REGION Network 34: PartExist
   RUNG wire#powerrail
      Contact( "AlwaysTRUE" )
      wire#w1
      Contact( "iF-ROOBT3Gripper1Detection" )
      Coil( "KukaRobot3_CtrlDB".sPLCtoROB.User.Gripper.DI133_PartOnGrip1 )
   END_RUNG
   RUNG wire#w1
      Contact( "iF-ROOBT3Gripper2Detection-" )
      Coil( "KukaRobot3_CtrlDB".sPLCtoROB.User.Gripper.DI134_PartOnGrip2 )
   END_RUNG
   // the same network as SCL:
   "KukaRobot3_CtrlDB".sPLCtoROB.User.Gripper.DI133_PartOnGrip1 := "AlwaysTRUE" AND "iF-ROOBT3Gripper1Detection";
   "KukaRobot3_CtrlDB".sPLCtoROB.User.Gripper.DI134_PartOnGrip2 := "AlwaysTRUE" AND "iF-ROOBT3Gripper2Detection-";
END_REGION

REGION Network 35: SpeedCount
   RUNG wire#powerrail
      Contact( "AlwaysTRUE" )
      wire#w1
      { S7_Templates := "SrcType := Int" } GE_Contact(in1 := "Robot_DB".Robot_3.SpeedCount, in2 := 2)
      Coil( "Robot_DB".Robot_3.SpeedChangeFlag )
   END_RUNG
   RUNG wire#w1
      I_Contact( "Station_Sys".Auto.Mode )
      Move(in := 0, out1 => "Robot_DB".Robot_3.SpeedCount)
   END_RUNG
   // the same network as SCL:
   "Robot_DB".Robot_3.SpeedChangeFlag := "AlwaysTRUE" AND ("Robot_DB".Robot_3.SpeedCount >= 2);
   IF "AlwaysTRUE" AND NOT "Station_Sys".Auto.Mode THEN "Robot_DB".Robot_3.SpeedCount := 0; END_IF;
END_REGION

REGION Network 36: Robot3Speed Interlock
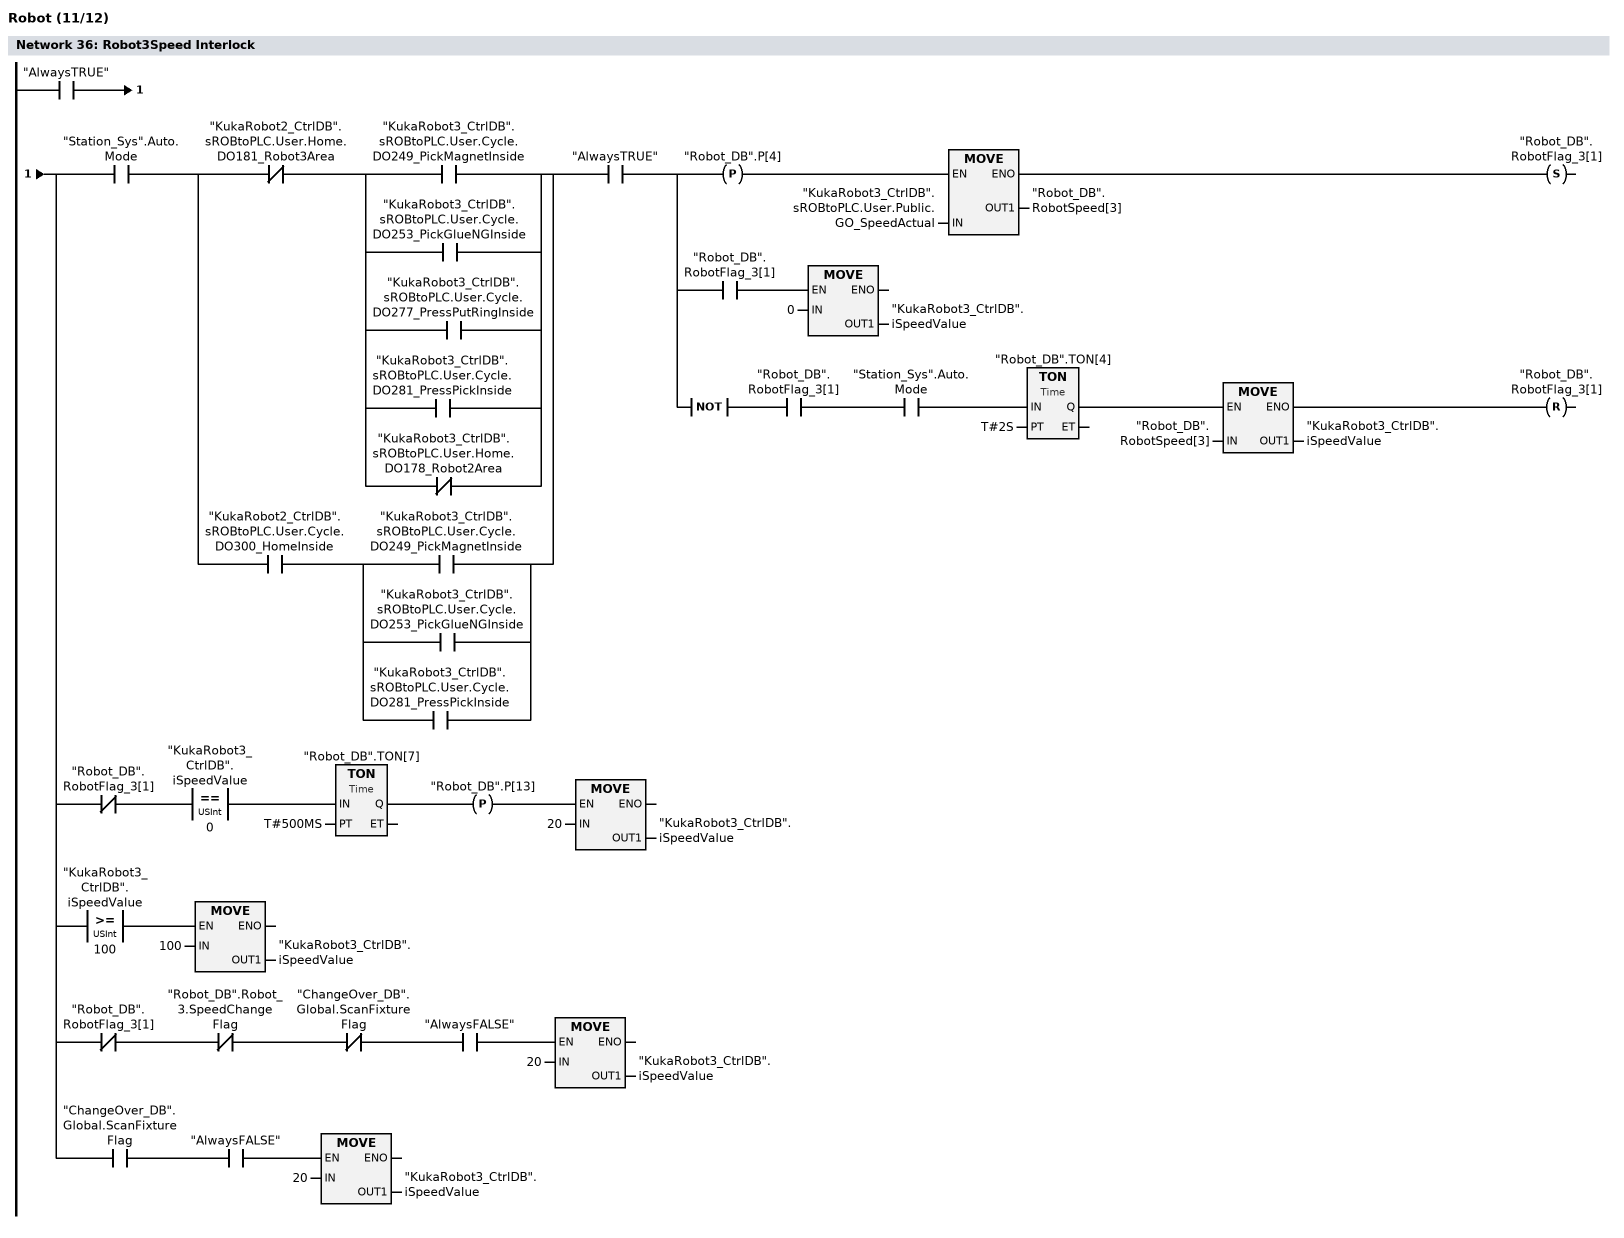
   RUNG wire#powerrail
      Contact( "AlwaysTRUE" )
      wire#w1
      Contact( "Station_Sys".Auto.Mode )
      wire#w2
      I_Contact( "KukaRobot2_CtrlDB".sROBtoPLC.User.Home.DO181_Robot3Area )
      wire#w3
      Contact( "KukaRobot3_CtrlDB".sROBtoPLC.User.Cycle.DO249_PickMagnetInside )
      wire#w4
      Contact( "AlwaysTRUE" )
      wire#w6
      P_Trig( "Robot_DB".P[4] )
      Move(in := "KukaRobot3_CtrlDB".sROBtoPLC.User.Public.GO_SpeedActual, out1 => "Robot_DB".RobotSpeed[3])
      S_Coil( "Robot_DB".RobotFlag_3[1] )
   END_RUNG
   RUNG wire#w3
      Contact( "KukaRobot3_CtrlDB".sROBtoPLC.User.Cycle.DO253_PickGlueNGInside )
   END_RUNG wire#w4
   RUNG wire#w3
      Contact( "KukaRobot3_CtrlDB".sROBtoPLC.User.Cycle.DO277_PressPutRingInside )
   END_RUNG wire#w4
   RUNG wire#w3
      Contact( "KukaRobot3_CtrlDB".sROBtoPLC.User.Cycle.DO281_PressPickInside )
   END_RUNG wire#w4
   RUNG wire#w3
      I_Contact( "KukaRobot3_CtrlDB".sROBtoPLC.User.Home.DO178_Robot2Area )
   END_RUNG wire#w4
   RUNG wire#w2
      Contact( "KukaRobot2_CtrlDB".sROBtoPLC.User.Cycle.DO300_HomeInside )
      wire#w5
      Contact( "KukaRobot3_CtrlDB".sROBtoPLC.User.Cycle.DO249_PickMagnetInside )
   END_RUNG wire#w4
   RUNG wire#w5
      Contact( "KukaRobot3_CtrlDB".sROBtoPLC.User.Cycle.DO253_PickGlueNGInside )
   END_RUNG wire#w4
   RUNG wire#w5
      Contact( "KukaRobot3_CtrlDB".sROBtoPLC.User.Cycle.DO281_PressPickInside )
   END_RUNG wire#w4
   RUNG wire#w6
      Contact( "Robot_DB".RobotFlag_3[1] )
      Move(in := 0, out1 => "KukaRobot3_CtrlDB".iSpeedValue)
   END_RUNG
   RUNG wire#w6
      Not()
      Contact( "Robot_DB".RobotFlag_3[1] )
      Contact( "Station_Sys".Auto.Mode )
      { S7_Templates := "time_type := Time" } "Robot_DB".TON[4].TON(pt := T#2S, et =>)
      Move(in := "Robot_DB".RobotSpeed[3], out1 => "KukaRobot3_CtrlDB".iSpeedValue)
      R_Coil( "Robot_DB".RobotFlag_3[1] )
   END_RUNG
   RUNG wire#w1
      I_Contact( "Robot_DB".RobotFlag_3[1] )
      { S7_Templates := "SrcType := USInt" } EQ_Contact(in1 := "KukaRobot3_CtrlDB".iSpeedValue, in2 := 0)
      { S7_Templates := "time_type := Time" } "Robot_DB".TON[7].TON(pt := T#500MS, et =>)
      P_Trig( "Robot_DB".P[13] )
      Move(in := 20, out1 => "KukaRobot3_CtrlDB".iSpeedValue)
   END_RUNG
   RUNG wire#w1
      { S7_Templates := "SrcType := USInt" } GE_Contact(in1 := "KukaRobot3_CtrlDB".iSpeedValue, in2 := 100)
      Move(in := 100, out1 => "KukaRobot3_CtrlDB".iSpeedValue)
   END_RUNG
   RUNG wire#w1
      I_Contact( "Robot_DB".RobotFlag_3[1] )
      I_Contact( "Robot_DB".Robot_3.SpeedChangeFlag )
      I_Contact( "ChangeOver_DB".Global.ScanFixtureFlag )
      Contact( "AlwaysFALSE" )
      Move(in := 20, out1 => "KukaRobot3_CtrlDB".iSpeedValue)
   END_RUNG
   RUNG wire#w1
      Contact( "ChangeOver_DB".Global.ScanFixtureFlag )
      Contact( "AlwaysFALSE" )
      Move(in := 20, out1 => "KukaRobot3_CtrlDB".iSpeedValue)
   END_RUNG
   // the same network as SCL:
   #_w1 := "AlwaysTRUE" AND "Station_Sys".Auto.Mode AND ((NOT "KukaRobot2_CtrlDB".sROBtoPLC.User.Home.DO181_Robot3Area AND ("KukaRobot3_CtrlDB".sROBtoPLC.User.Cycle.DO249_PickMagnetInside OR "KukaRobot3_CtrlDB".sROBtoPLC.User.Cycle.DO253_PickGlueNGInside OR "KukaRobot3_CtrlDB".sROBtoPLC.User.Cycle.DO277_PressPutRingInside OR "KukaRobot3_CtrlDB".sROBtoPLC.User.Cycle.DO281_PressPickInside OR NOT "KukaRobot3_CtrlDB".sROBtoPLC.User.Home.DO178_Robot2Area)) OR ("KukaRobot2_CtrlDB".sROBtoPLC.User.Cycle.DO300_HomeInside AND ("KukaRobot3_CtrlDB".sROBtoPLC.User.Cycle.DO249_PickMagnetInside OR "KukaRobot3_CtrlDB".sROBtoPLC.User.Cycle.DO253_PickGlueNGInside OR "KukaRobot3_CtrlDB".sROBtoPLC.User.Cycle.DO281_PressPickInside))) AND "AlwaysTRUE";
   #_w2 := #_w1 AND NOT "Robot_DB".P[4];   // rising edge
   "Robot_DB".P[4] := #_w1;
   IF #_w2 THEN
       "Robot_DB".RobotSpeed[3] := "KukaRobot3_CtrlDB".sROBtoPLC.User.Public.GO_SpeedActual;
       "Robot_DB".RobotFlag_3[1] := TRUE;
   END_IF;
   IF #_w1 AND "Robot_DB".RobotFlag_3[1] THEN "KukaRobot3_CtrlDB".iSpeedValue := 0; END_IF;
   "Robot_DB".TON[4].TON(IN := NOT #_w1 AND "Robot_DB".RobotFlag_3[1] AND "Station_Sys".Auto.Mode, PT := T#2S);
   IF "Robot_DB".TON[4].Q THEN
       "KukaRobot3_CtrlDB".iSpeedValue := "Robot_DB".RobotSpeed[3];
       "Robot_DB".RobotFlag_3[1] := FALSE;
   END_IF;
   "Robot_DB".TON[7].TON(IN := "AlwaysTRUE" AND NOT "Robot_DB".RobotFlag_3[1] AND ("KukaRobot3_CtrlDB".iSpeedValue = 0),
                         PT := T#500MS);
   #_w3 := "Robot_DB".TON[7].Q AND NOT "Robot_DB".P[13];   // rising edge
   "Robot_DB".P[13] := "Robot_DB".TON[7].Q;
   IF #_w3 THEN "KukaRobot3_CtrlDB".iSpeedValue := 20; END_IF;
   IF "AlwaysTRUE" AND ("KukaRobot3_CtrlDB".iSpeedValue >= 100) THEN
       "KukaRobot3_CtrlDB".iSpeedValue := 100;
   END_IF;
   IF "AlwaysTRUE" AND NOT "Robot_DB".RobotFlag_3[1] AND NOT "Robot_DB".Robot_3.SpeedChangeFlag AND NOT "ChangeOver_DB".Global.ScanFixtureFlag AND "AlwaysFALSE" THEN
       "KukaRobot3_CtrlDB".iSpeedValue := 20;
   END_IF;
   IF "AlwaysTRUE" AND "ChangeOver_DB".Global.ScanFixtureFlag AND "AlwaysFALSE" THEN
       "KukaRobot3_CtrlDB".iSpeedValue := 20;
   END_IF;
END_REGION

REGION Network 37: Robot3 No Task Running
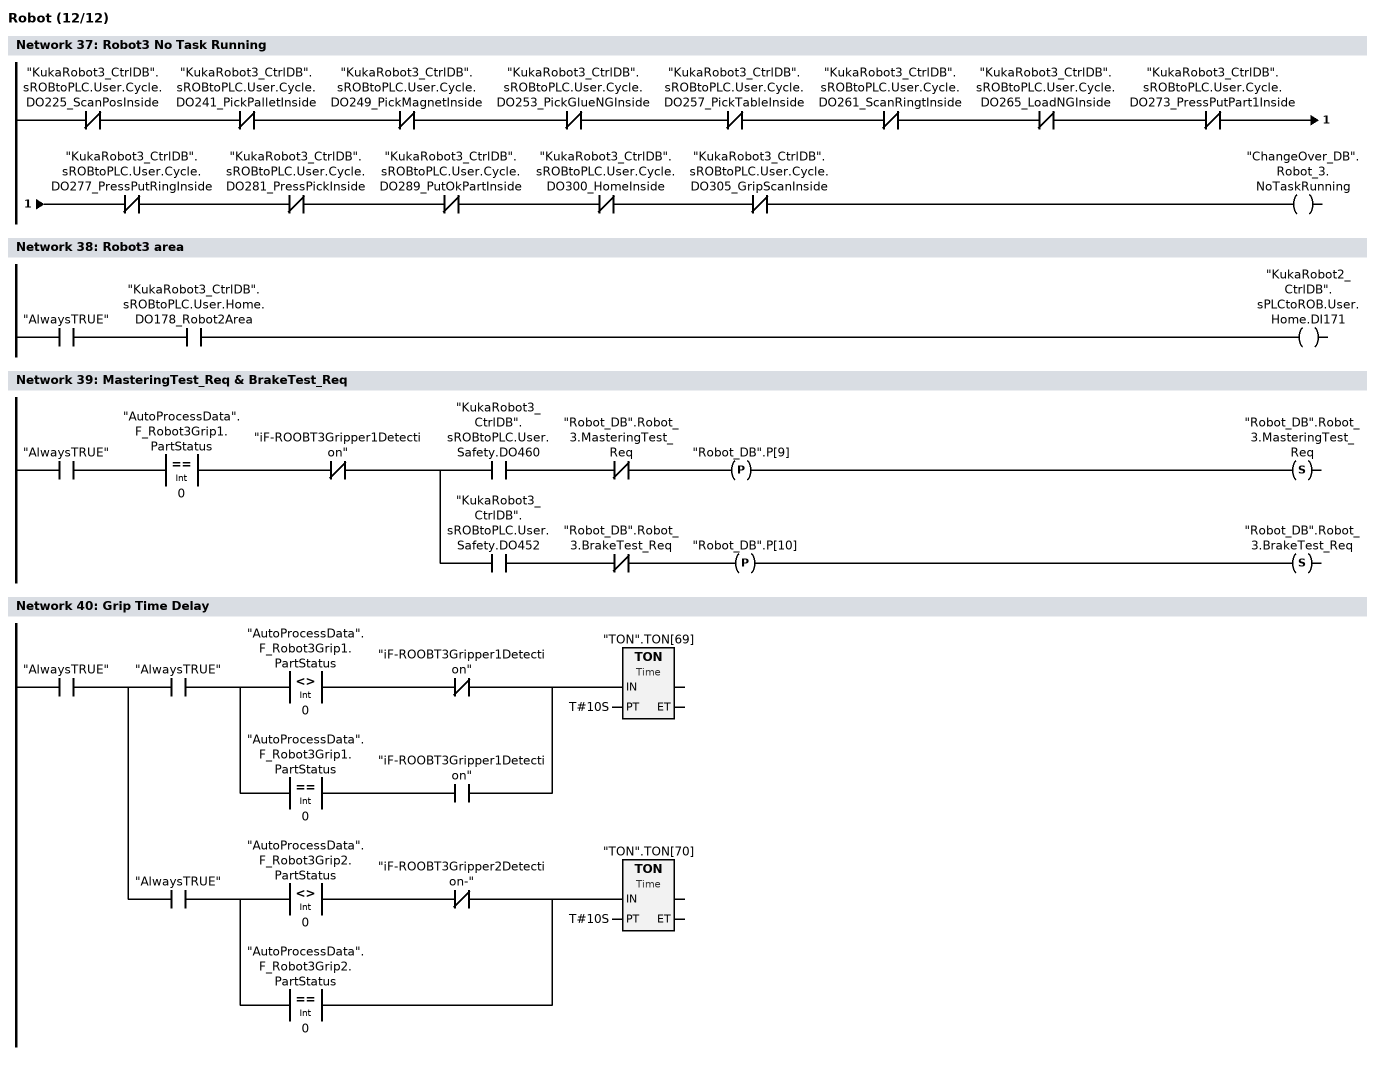
   RUNG wire#powerrail
      I_Contact( "KukaRobot3_CtrlDB".sROBtoPLC.User.Cycle.DO225_ScanPosInside )
      I_Contact( "KukaRobot3_CtrlDB".sROBtoPLC.User.Cycle.DO241_PickPalletInside )
      I_Contact( "KukaRobot3_CtrlDB".sROBtoPLC.User.Cycle.DO249_PickMagnetInside )
      I_Contact( "KukaRobot3_CtrlDB".sROBtoPLC.User.Cycle.DO253_PickGlueNGInside )
      I_Contact( "KukaRobot3_CtrlDB".sROBtoPLC.User.Cycle.DO257_PickTableInside )
      I_Contact( "KukaRobot3_CtrlDB".sROBtoPLC.User.Cycle.DO261_ScanRingtInside )
      I_Contact( "KukaRobot3_CtrlDB".sROBtoPLC.User.Cycle.DO265_LoadNGInside )
      I_Contact( "KukaRobot3_CtrlDB".sROBtoPLC.User.Cycle.DO273_PressPutPart1Inside )
      I_Contact( "KukaRobot3_CtrlDB".sROBtoPLC.User.Cycle.DO277_PressPutRingInside )
      I_Contact( "KukaRobot3_CtrlDB".sROBtoPLC.User.Cycle.DO281_PressPickInside )
      I_Contact( "KukaRobot3_CtrlDB".sROBtoPLC.User.Cycle.DO289_PutOkPartInside )
      I_Contact( "KukaRobot3_CtrlDB".sROBtoPLC.User.Cycle.DO300_HomeInside )
      I_Contact( "KukaRobot3_CtrlDB".sROBtoPLC.User.Cycle.DO305_GripScanInside )
      Coil( "ChangeOver_DB".Robot_3.NoTaskRunning )
   END_RUNG
   // the same network as SCL:
   "ChangeOver_DB".Robot_3.NoTaskRunning := NOT "KukaRobot3_CtrlDB".sROBtoPLC.User.Cycle.DO225_ScanPosInside AND NOT "KukaRobot3_CtrlDB".sROBtoPLC.User.Cycle.DO241_PickPalletInside AND NOT "KukaRobot3_CtrlDB".sROBtoPLC.User.Cycle.DO249_PickMagnetInside AND NOT "KukaRobot3_CtrlDB".sROBtoPLC.User.Cycle.DO253_PickGlueNGInside AND NOT "KukaRobot3_CtrlDB".sROBtoPLC.User.Cycle.DO257_PickTableInside AND NOT "KukaRobot3_CtrlDB".sROBtoPLC.User.Cycle.DO261_ScanRingtInside AND NOT "KukaRobot3_CtrlDB".sROBtoPLC.User.Cycle.DO265_LoadNGInside AND NOT "KukaRobot3_CtrlDB".sROBtoPLC.User.Cycle.DO273_PressPutPart1Inside AND NOT "KukaRobot3_CtrlDB".sROBtoPLC.User.Cycle.DO277_PressPutRingInside AND NOT "KukaRobot3_CtrlDB".sROBtoPLC.User.Cycle.DO281_PressPickInside AND NOT "KukaRobot3_CtrlDB".sROBtoPLC.User.Cycle.DO289_PutOkPartInside AND NOT "KukaRobot3_CtrlDB".sROBtoPLC.User.Cycle.DO300_HomeInside AND NOT "KukaRobot3_CtrlDB".sROBtoPLC.User.Cycle.DO305_GripScanInside;
END_REGION

REGION Network 38: Robot3 area
   RUNG wire#powerrail
      Contact( "AlwaysTRUE" )
      Contact( "KukaRobot3_CtrlDB".sROBtoPLC.User.Home.DO178_Robot2Area )
      Coil( "KukaRobot2_CtrlDB".sPLCtoROB.User.Home.DI171 )
   END_RUNG
   // the same network as SCL:
   "KukaRobot2_CtrlDB".sPLCtoROB.User.Home.DI171 := "AlwaysTRUE" AND "KukaRobot3_CtrlDB".sROBtoPLC.User.Home.DO178_Robot2Area;
END_REGION

REGION Network 39: MasteringTest_Req & BrakeTest_Req
   RUNG wire#powerrail
      Contact( "AlwaysTRUE" )
      { S7_Templates := "SrcType := Int" } EQ_Contact(in1 := "AutoProcessData".F_Robot3Grip1.PartStatus, in2 := 0)
      I_Contact( "iF-ROOBT3Gripper1Detection" )
      wire#w1
      Contact( "KukaRobot3_CtrlDB".sROBtoPLC.User.Safety.DO460 )
      I_Contact( "Robot_DB".Robot_3.MasteringTest_Req )
      P_Trig( "Robot_DB".P[9] )
      S_Coil( "Robot_DB".Robot_3.MasteringTest_Req )
   END_RUNG
   RUNG wire#w1
      Contact( "KukaRobot3_CtrlDB".sROBtoPLC.User.Safety.DO452 )
      I_Contact( "Robot_DB".Robot_3.BrakeTest_Req )
      P_Trig( "Robot_DB".P[10] )
      S_Coil( "Robot_DB".Robot_3.BrakeTest_Req )
   END_RUNG
   // the same network as SCL:
   #_w1 := "AlwaysTRUE" AND ("AutoProcessData".F_Robot3Grip1.PartStatus = 0) AND NOT "iF-ROOBT3Gripper1Detection";
   #_w2 := #_w1 AND "KukaRobot3_CtrlDB".sROBtoPLC.User.Safety.DO460 AND NOT "Robot_DB".Robot_3.MasteringTest_Req;
   #_w3 := #_w2 AND NOT "Robot_DB".P[9];   // rising edge
   "Robot_DB".P[9] := #_w2;
   IF #_w3 THEN "Robot_DB".Robot_3.MasteringTest_Req := TRUE; END_IF;
   #_w4 := #_w1 AND "KukaRobot3_CtrlDB".sROBtoPLC.User.Safety.DO452 AND NOT "Robot_DB".Robot_3.BrakeTest_Req;
   #_w5 := #_w4 AND NOT "Robot_DB".P[10];   // rising edge
   "Robot_DB".P[10] := #_w4;
   IF #_w5 THEN "Robot_DB".Robot_3.BrakeTest_Req := TRUE; END_IF;
END_REGION

REGION Network 40: Grip Time Delay
   RUNG wire#powerrail
      Contact( "AlwaysTRUE" )
      wire#w1
      Contact( "AlwaysTRUE" )
      wire#w2
      { S7_Templates := "SrcType := Int" } NE_Contact(in1 := "AutoProcessData".F_Robot3Grip1.PartStatus, in2 := 0)
      I_Contact( "iF-ROOBT3Gripper1Detection" )
      wire#w3
      { S7_Templates := "time_type := Time" } "TON".TON[69].TON(pt := T#10S, et =>)
   END_RUNG
   RUNG wire#w2
      { S7_Templates := "SrcType := Int" } EQ_Contact(in1 := "AutoProcessData".F_Robot3Grip1.PartStatus, in2 := 0)
      Contact( "iF-ROOBT3Gripper1Detection" )
   END_RUNG wire#w3
   RUNG wire#w1
      Contact( "AlwaysTRUE" )
      wire#w4
      { S7_Templates := "SrcType := Int" } NE_Contact(in1 := "AutoProcessData".F_Robot3Grip2.PartStatus, in2 := 0)
      I_Contact( "iF-ROOBT3Gripper2Detection-" )
      wire#w5
      { S7_Templates := "time_type := Time" } "TON".TON[70].TON(pt := T#10S, et =>)
   END_RUNG
   RUNG wire#w4
      { S7_Templates := "SrcType := Int" } EQ_Contact(in1 := "AutoProcessData".F_Robot3Grip2.PartStatus, in2 := 0)
   END_RUNG wire#w5
   // the same network as SCL:
   "TON".TON[69].TON(IN := "AlwaysTRUE" AND "AlwaysTRUE" AND ((("AutoProcessData".F_Robot3Grip1.PartStatus <> 0) AND NOT "iF-ROOBT3Gripper1Detection") OR (("AutoProcessData".F_Robot3Grip1.PartStatus = 0) AND "iF-ROOBT3Gripper1Detection")),
                     PT := T#10S);
   "TON".TON[70].TON(IN := "AlwaysTRUE" AND "AlwaysTRUE" AND ((("AutoProcessData".F_Robot3Grip2.PartStatus <> 0) AND NOT "iF-ROOBT3Gripper2Detection-") OR ("AutoProcessData".F_Robot3Grip2.PartStatus = 0)),
                     PT := T#10S);
END_REGION
END_FUNCTION

FUNCTION_BLOCK "KukaRobot1_Ctrl"   // FB2401, SCL
{ S7_Optimized_Access := 'FALSE' }
// stored: AutoNumber false, SetENOAutomatically false
   VAR_INPUT
      iHWID_In : HW_IO;
      iHWID_Out : HW_IO;
      iSysRun : Bool;
      iAuto : Bool;
      iManual : Bool;
      iSpecial : Bool;
      iE_STOP : Bool;
      iReset : Bool;
      iT1000ms : Bool;
      iTaskMode : USInt;
      iPartType : USInt;
      iSpeedValue : USInt;
      iPGNO : USInt;   // Robot Program number
   END_VAR
   VAR_OUTPUT
      oReady : Bool;
      oStartComplete : Bool;
      oWarning : Bool;
      oError : Bool;
      oErrorCode : Int;
   END_VAR
   VAR_IN_OUT
      ioAutoStart : Bool;
      ioSrartHome : Bool;
      ioStartAutoCycle : Bool;
   END_VAR
   VAR
      sHMI { S7_SetPoint := 'True'} : "KukaRobot_HMI";
      sROBtoPLC : Struct
         Sys { S7_SetPoint := 'True'} : "KukaRobot_SysOutput";   // Robot ---> PLC
         User { S7_SetPoint := 'True'} : "KukaRobot_UserOutput_1";   // Robot ---> PLC
      END_STRUCT;
      sPLCtoROB : Struct
         Sys { S7_SetPoint := 'True'} : "KukaRobot_SysInput";   // PLC ---> Robot
         User { S7_SetPoint := 'True'} : "KukaRobot_UserInput_1";   // PLC ---> Robot
      END_STRUCT;
      sDrivesOnDelay { S7_SetPoint := 'True'} : TON_TIME;
      sStartUpDelay { S7_SetPoint := 'True'} : TON_TIME;
      sRobotReadyToStart : Bool;
      sRobotReadyToRunning : Bool;
      sRobotActComplete : Bool;
      sRobotProgrameChoseOK : Bool;
      sSequence : Int;
      F_TRIG_Work { S7_SetPoint := 'True'} : F_TRIG;
      F_TRIG_Home { S7_SetPoint := 'True'} : F_TRIG;
      ModeValue : Int;
      Tem_ModeValue : Int;
      ModeChange : Bool;
      IEC_Timer_DRIVES_OFF { S7_SetPoint := 'True'} : TON_TIME;
      IEC_Timer_DRIVES_ON { S7_SetPoint := 'True'} : TON_TIME;
   END_VAR
   VAR_TEMP
      tInRwENO : Bool;
      tOutRwENO : Bool;
      tInRwRetVal : Int;
      tOutRwRetVal : Int;
      "tROB-Input" : Array[1..128] of Byte;
      tROB_Output : Array[1..128] of Byte;
   END_VAR
BEGIN
   REGION Description
       (*
       %%%
   VERSION: V1.0
   LANGUAGE: ENGLISH
       %%%
       ** ** ** ** ** ** ** ** ** ** ** ** ** ** ** ** ** ** ** ** ** ** ** ** ** ** ** ** ** ** ** ** ** ** ** ** ** ** ** ** ** ** ** ** ** ** ** ** ** **
       ** ** ** ** ** ** ** ** ** ** ** ** ** ** ** ** ** ** ** ** ** ** ** ** ** ** ** ** ** ** ** ** ** ** ** ** ** ** ** ** ** ** ** ** ** ** ** ** ** **
       * *
       * R (uhlamat) R (obot) I (nterface) *
       * < < Robot Function Block > > *
       * < < Handing Tool > > *
       * - - - - - - - - - - - - - - - - - - - - - - - - - - - - - - - - - - - - - - - - - - *
       * *
       * Customer:   *
       * Roboter Type: Kuka *
       * Software: Siemens TIA V15.1 SP1 *
       * Autor: ChenYi *
       * Company: Ruhlamat Automation Technologies (Suzhou) Co., Ltd *
       * Department: Elec.*
       * Telephone: + 86 (512) 6767 1108 *
       * *
       * Version: 1.0 *
       * Created: 26.05.2020 *
       * Modified: 26.05.2020
   BY: ChenYi *
       * *
       ** ** ** ** ** ** ** ** ** ** ** ** ** ** ** ** ** ** ** ** ** ** ** ** ** ** ** ** ** ** ** ** ** ** ** ** ** ** ** ** ** ** ** ** ** ** ** ** ** **
       ** ** ** ** ** ** ** ** ** ** ** ** ** ** ** ** ** ** ** ** ** ** ** ** ** ** ** ** ** ** ** ** ** ** ** ** ** ** ** ** ** ** ** ** ** ** ** ** ** **
       %%%
    #oErrorCode:
       102:Robot home Failed
       205:Failed to read HW Input data;
       206:Failed to write HW Output data;
       303:Start up TimeOut   

       %%%
       *)
   END_REGION
   //<<<<<<<<<<<<<<<<<<<<<<<<<<<<<<<<<<<<<<<<<<<<<<<<<>>>>>>>>>>>>>>>>>>>>>>>>>>>>>>>>>>>>>>>>>>>>>>>>>
   //<<<<<<<<<<<<<<<<<<<<<<<<<<<<<<<<<<<<<<<<  Program Start  >>>>>>>>>>>>>>>>>>>>>>>>>>>>>>>>>>>>>>>>>
   //<<<<<<<<<<<<<<<<<<<<<<<<<<<<<<<<<<<<<<<<<<<<<<<<<>>>>>>>>>>>>>>>>>>>>>>>>>>>>>>>>>>>>>>>>>>>>>>>>>




   //******************************************
   REGION Bus Input Data Mapping

       #tInRwRetVal := DPRD_DAT(LADDR := #iHWID_In, RECORD => #sROBtoPLC, ENO => #tInRwENO);
       IF NOT #tInRwENO THEN
           GOTO ERROR;
       END_IF;

   END_REGION


   //******************************************
   (*Robot controller remmote control*)

   // I/O Act-Activate interface
   #sPLCtoROB.Sys.SI.I_O_ACT := 1;
   // Move Enable
   //#sPLCtoROB.Sys.SI.MOVE_ENABLE := (#iSysRun AND (((#sROBtoPLC.Sys.SO.T1 OR #sROBtoPLC.Sys.SO.T2) AND #iManual) OR (#iAuto))) AND #iSafePos;
   //#sPLCtoROB.Sys.SI.MOVE_ENABLE := #iSysRun AND (#iManual OR #iAuto) AND #iSafePos;
   IF #sROBtoPLC.Sys.SO.EXT = TRUE THEN
       #sPLCtoROB.Sys.SI.MOVE_ENABLE := #iE_STOP;
   END_IF;
   IF #sROBtoPLC.Sys.SO.T1 = TRUE OR #sROBtoPLC.Sys.SO.T2 = TRUE THEN
       #sPLCtoROB.Sys.SI.MOVE_ENABLE := TRUE;
   END_IF;
   // Drives Off
   #sPLCtoROB.Sys.SI.DRIVES_OFF := NOT #ModeChange;


   IF #iManual
   THEN
       #ModeValue := 1;
   ELSIF #iAuto
   THEN
       #ModeValue := 3;

   END_IF;

   IF #ModeValue <> #Tem_ModeValue
   THEN
       #ModeChange := true;
   ELSE
       #ModeChange := false;
   END_IF;

   IF #IEC_Timer_DRIVES_OFF.Q THEN
       #Tem_ModeValue := #ModeValue;
   END_IF;

   #IEC_Timer_DRIVES_OFF(IN:=#ModeValue <> #Tem_ModeValue,
                         PT:=T#1s);


   //#sPLCtoROB.Sys.SI.DRIVES_OFF := #iSysRun;
   //#sPLCtoROB.Sys.SI.DRIVES_OFF := #iSysRun AND (#iManual OR #iAuto) AND #iSafePos;
   (*Robot controller ready to Start*)
   #sRobotReadyToStart := #iSysRun AND (#iAuto OR #iSpecial) AND
   #sROBtoPLC.Sys.SO.USER_SAF AND #sROBtoPLC.Sys.SO.ALARM_STOP AND
   #sROBtoPLC.Sys.SO.I_O_ACTCONF AND #sROBtoPLC.Sys.SO.ALARM_STOP_INTERN AND
   #sPLCtoROB.Sys.SI.MOVE_ENABLE AND #sPLCtoROB.Sys.SI.DRIVES_OFF
   AND #sROBtoPLC.Sys.SO.EXT;


   REGION Robot Start control
       IF #sRobotReadyToStart THEN
           IF (#sSequence = 0) AND #ioAutoStart AND (#iAuto OR #iSpecial) AND NOT #sRobotActComplete THEN
               #sSequence := 100;
               #ioAutoStart := 0;
               #sRobotActComplete := 0;
               #sRobotProgrameChoseOK := 0;
           END_IF;

           #IEC_Timer_DRIVES_ON(IN := #sSequence=110,
                                 PT := T#100ms);

           CASE #sSequence OF
   (*            100:
                   #sPLCtoROB.Sys.SI.DRIVES_ON := 0;
                   #sSequence := 110;

               110:
                   #sPLCtoROB.Sys.SI.DRIVES_ON := 1;
                   IF #IEC_Timer_DRIVES_ON.Q THEN
                       #sPLCtoROB.Sys.SI.DRIVES_ON := 0;
                       #sSequence := 150;
                   END_IF;
                   *)
               100:  // DrivesOn
                   IF NOT #sROBtoPLC.Sys.SO.RC_RDY1  THEN
                           #sPLCtoROB.Sys.SI.CONF_MESS := 1;
                           #sPLCtoROB.Sys.SI.DRIVES_ON := 0;
                       ELSIF #sROBtoPLC.Sys.SO.RC_RDY1 THEN
                           #sPLCtoROB.Sys.SI.CONF_MESS := 0;
                           #sPLCtoROB.Sys.SI.DRIVES_ON := 1;
                           IF #sDrivesOnDelay.Q AND #sROBtoPLC.Sys.SO.PERI_RDY THEN
                               #sSequence := 200;
                               #sPLCtoROB.Sys.SI.DRIVES_ON := 0;

                           END_IF;
                       END_IF;

                       200:  // ALARM CONF
                       IF #sROBtoPLC.Sys.SO.STOPMESS OR NOT #sROBtoPLC.Sys.SO.RC_RDY1 THEN
                           #sPLCtoROB.Sys.SI.CONF_MESS := 1;
                       ELSE
                           #sPLCtoROB.Sys.SI.CONF_MESS := 0;
                           #sSequence := 300;
                       END_IF;

                       300: // EXT_Start    
                       IF #sROBtoPLC.Sys.SO.PERI_RDY AND NOT #sROBtoPLC.Sys.SO.STOPMESS THEN
                           #sPLCtoROB.Sys.SI.EXT_START := 1;
                           #sSequence := 400;
                       END_IF;

                       400: // EXT_Start Reset  
                       IF #sROBtoPLC.Sys.SO.PRO_ACT THEN
                           #sPLCtoROB.Sys.SI.EXT_START := 0;
                           #sSequence := 500;
                       END_IF;

                       500: // Programe Call
                       IF #sROBtoPLC.Sys.SO.PERI_RDY
                           AND #sROBtoPLC.Sys.SO.PRO_ACT
                           AND #sROBtoPLC.Sys.SO.PGNO_REQ
                           AND #iPGNO <> 0
                           //AND #s_ROBInput.User.User.Home.DI_AutoCycleStart
                           //AND #s_ROBOutput.Sys."SO_$ON_PATH"
                           //AND #s_ROBOutput.Sys."SO_$IN_HOME"
                       THEN

                           #sPLCtoROB.Sys.SI.PGNO_PBIT := #iPGNO;
                           #sPLCtoROB.Sys.SI.PGNO_VALID := 1;
                           #sSequence := 600;
                       END_IF;

                       600: // Programe Call Finish
                       IF #sROBtoPLC.Sys.SO.APPL_RUN THEN
                           #sPLCtoROB.Sys.SI.PGNO_VALID := 0;
                           #sRobotActComplete := 1;
                           #sSequence := 0;
                       END_IF;

           END_CASE;

       ELSE
           #sSequence := 0;
           #sRobotActComplete := 0;
   //        #sPLCtoROB.Sys.SI.DRIVES_ON := 0;////2023/9/1更改
           #sPLCtoROB.Sys.SI.EXT_START := 0;
          // #sPLCtoROB.Sys.SI.CONF_MESS := 0;
           #sPLCtoROB.Sys.SI.PGNO_VALID := 0;
           #sPLCtoROB.Sys.SI.PGNO_PBIT := 0; 
       END_IF;

   (*Robot ready to Running*)
       #sRobotReadyToRunning := #sRobotReadyToStart AND #sROBtoPLC.Sys.SO.PERI_RDY AND #sROBtoPLC.Sys.SO.PRO_ACT AND #sROBtoPLC.Sys.SO.APPL_RUN;


   (*Robot TaskMode,PartType, SpeedValue Set*)
       #sPLCtoROB.User.Public.GI_TaskMode := #iTaskMode;
       #sPLCtoROB.User.Public.GI_PartType := #iPartType;
       #sPLCtoROB.User.Public.GI_SpeedSet := #iSpeedValue;

       // Robot Program calls
       #sPLCtoROB.Sys.SI.PGNO_PARITY := 1;
       //************************************************************
       (*DrivesOn delay*)
       #sDrivesOnDelay(IN := #sPLCtoROB.Sys.SI.DRIVES_ON,
                       PT := T#200ms      // IN: TIME
       );
   (*StartTimeOut delay*)
       #sStartUpDelay(IN := #sSequence <> 0,
                      PT := T#5s        // IN: TIME
       );
       IF #sStartUpDelay.Q THEN
           #sHMI.StartUpTimeOut := 1;
           GOTO ERROR;
       ELSE
           #sHMI.StartUpTimeOut := 0;
       END_IF;

   END_REGION

   //******************************************
   REGION Home
       IF #sRobotReadyToRunning AND #sROBtoPLC.User.Home.DO161_WaitForHomeSeqStart AND NOT #sROBtoPLC.User.Home.DO162_GoHomeFail AND #ioSrartHome THEN
           #sPLCtoROB.User.Home.DI161_HomeSeqStart := 1;
       END_IF;

       IF #sRobotReadyToRunning AND #sROBtoPLC.User.Home.DO163_HomeSeqOK THEN
           #ioSrartHome := 0;
           #sPLCtoROB.User.Home.DI161_HomeSeqStart := 0;
       END_IF;

       IF #sROBtoPLC.User.Home.DO162_GoHomeFail THEN
           GOTO ERROR;
       END_IF;

   END_REGION ;

   REGION Auto Cycle Start

       (*Start Auto Cycle*)
       IF #sRobotReadyToRunning AND #sROBtoPLC.User.Home.DO164_WaitForAutoStart AND #ioStartAutoCycle THEN
           #sPLCtoROB.User.Home.DI162_AutoCycleStart := 1;
       ELSE
           #sPLCtoROB.User.Home.DI162_AutoCycleStart := 0;
       END_IF;

       IF NOT #sROBtoPLC.User.Home.DO164_WaitForAutoStart THEN
           #ioStartAutoCycle := 0;
       END_IF;


   END_REGION ;




   REGION Bus Output Data Mapping

       #tOutRwRetVal := DPWR_DAT(LADDR := #iHWID_Out, RECORD := #sPLCtoROB, ENO => #tOutRwENO);
       IF NOT #tOutRwENO THEN
           GOTO ERROR;
       END_IF;

   END_REGION

   //----------------------------------------------------------------------------------------------------
   REGION Output
       #oReady := #sRobotReadyToRunning;
       #oStartComplete := #sRobotActComplete;


   END_REGION

   REGION HMI Signal
       //SI  
       #sHMI.PGNO_PBIT := #sPLCtoROB.Sys.SI.PGNO_PBIT;
       #sHMI.EXT_START := #sPLCtoROB.Sys.SI.EXT_START;
       #sHMI.MOVE_ENABLE := #sHMI.MOVE_ENABLE;
       #sHMI.CONF_MESS := #sPLCtoROB.Sys.SI.CONF_MESS;
       #sHMI.DRIVES_OFF := NOT #sHMI.DRIVES_OFF;
       #sHMI.DRIVES_ON := #sHMI.DRIVES_ON;
       #sHMI.I_O_ACT := #sHMI.I_O_ACT;
       //UI   
       #sHMI.TaskMode := #sPLCtoROB.User.Public.GI_TaskMode;
       #sHMI.PartType := #sPLCtoROB.User.Public.GI_PartType;
       #sHMI.SpeedSet := #sPLCtoROB.User.Public.GI_SpeedSet;
       #sHMI.HomeSeqStart := #sPLCtoROB.User.Home.DI161_HomeSeqStart;
       #sHMI.AutoCycleStart := #sPLCtoROB.User.Home.DI162_AutoCycleStart;
       //SO   
       #sHMI.RC_RDY1 := #sROBtoPLC.Sys.SO.RC_RDY1;
       #sHMI.ALARM_STOP := NOT #sROBtoPLC.Sys.SO.ALARM_STOP;
       #sHMI.USER_SAF := #sROBtoPLC.Sys.SO.USER_SAF;
       #sHMI.PERI_RDY := #sROBtoPLC.Sys.SO.PERI_RDY;
       #sHMI.ROB_CAL := #sROBtoPLC.Sys.SO.ROB_CAL;
       #sHMI.I_O_ACTCONF := #sROBtoPLC.Sys.SO.I_O_ACTCONF;
       #sHMI.STOPMESS := #sROBtoPLC.Sys.SO.STOPMESS;
       #sHMI.ALARM_STOP_INTERN := NOT #sROBtoPLC.Sys.SO.ALARM_STOP_INTERN;
       #sHMI.PGNO_FBIT_REFL := #sROBtoPLC.Sys.SO.PGNO_FBIT_REFL;
       #sHMI.PRO_ACT := #sROBtoPLC.Sys.SO.PRO_ACT;
       #sHMI.APPL_RUN := #sROBtoPLC.Sys.SO.APPL_RUN;
       #sHMI.PRO_MOVE := #sROBtoPLC.Sys.SO.PRO_MOVE;
       #sHMI.IN_HOME := #sROBtoPLC.Sys.SO.IN_HOME;
       #sHMI.ON_PATH := #sROBtoPLC.Sys.SO.ON_PATH;
       #sHMI.NEAR_POSRET := #sROBtoPLC.Sys.SO.NEAR_POSRET;
       #sHMI.T1 := #sROBtoPLC.Sys.SO.T1;
       #sHMI.T2 := #sROBtoPLC.Sys.SO.T2;
       #sHMI.AUT := #sROBtoPLC.Sys.SO.AUT;
       #sHMI.EXT := #sROBtoPLC.Sys.SO.EXT;
       //UO
       #sHMI.CurrentMode := #sROBtoPLC.User.Public.GO_CurrentMode;
       #sHMI.CurrentPartType := #sROBtoPLC.User.Public.GO_CurrentPartType;
       #sHMI.SpeedActual := #sROBtoPLC.User.Public.GO_SpeedActual;
       #sHMI.ProgramSequence := #sROBtoPLC.User.Public.GO_RobotTaskSequence;
       #sHMI.WaitForHomeSeqStart := #sROBtoPLC.User.Home.DO161_WaitForHomeSeqStart;
       #sHMI.GoHomeFail := #sROBtoPLC.User.Home.DO162_GoHomeFail;
       #sHMI.HomeSeqOK := #sROBtoPLC.User.Home.DO163_HomeSeqOK;
       #sHMI.WaitForAutoCycleStart := #sROBtoPLC.User.Home.DO164_WaitForAutoStart;
       //IO
       #sHMI.iTaskMode := #iTaskMode;
       #sHMI.iPartType := #iPartType;
       #sHMI.iSpeedValue := #iSpeedValue;
       #sHMI.iPGNO := #iPGNO;

       #sHMI.AutoStart := #ioAutoStart;
       #sHMI.SrartHome := #ioSrartHome;
       #sHMI.StartAutoCycle := #ioStartAutoCycle;

       #sHMI.Ready := #oReady;
       #sHMI.StartComplete := #oStartComplete;
       #sHMI.Warning := #oWarning;


   (*Robot working time monitor*)
       IF #iT1000ms AND NOT #sHMI.CountPulse AND #sROBtoPLC.Sys.SO.PERI_RDY THEN
           #sHMI.Seconds := #sHMI.Seconds + 1;
       END_IF;
       #sHMI.CountPulse := #iT1000ms;
       IF #sHMI.Seconds >= 60 THEN
           #sHMI.Minute := #sHMI.Minute + 1;
           #sHMI.Seconds := 0;
       END_IF;
       IF #sHMI.Minute >= 60 THEN
           #sHMI.Hours := #sHMI.Hours + 1;
           #sHMI.Minute := 0;
       END_IF;

   END_REGION

   REGION Error

       IF #iReset AND #oError THEN
           #oError := FALSE;
           #oErrorCode := 0;
       END_IF;

   ERROR:
       ENO := 0;

       IF #sROBtoPLC.User.Home.DO162_GoHomeFail THEN
           #oErrorCode := 102;
       ELSIF #tInRwRetVal <> 0 OR NOT #tInRwENO THEN
           #oError := 1;
           #oErrorCode := 205;
       ELSIF #tOutRwRetVal <> 0 OR NOT #tOutRwENO THEN
           #oError := 1;
           #oErrorCode := 206;
       ELSIF #sStartUpDelay.Q THEN
           #oError := 1;
           #oErrorCode := 303;
       END_IF;



       #sHMI.Error := #oError;
       #sHMI.ErrorCode := #oErrorCode;


   END_REGION

   // IF #sROBtoPLC.User.Gripper.DO129_GripperOpen THEN
   //     "ST10Cylinder".Cy[13].Inout.ManualGoHome := TRUE;
   //     "ST10Cylinder".Cy[13].Inout.ManualGoWork := FALSE;
   // END_IF;

   // IF #sROBtoPLC.User.Gripper.DO130_GripperClose THEN
   //     "ST10Cylinder".Cy[13].Inout.ManualGoWork := TRUE;
   //     "ST10Cylinder".Cy[13].Inout.ManualGoHome := FALSE;
   // END_IF;

   // #F_TRIG_Work(CLK:=#sROBtoPLC.User.Gripper.DO130_GripperClose);

   // #F_TRIG_Home(CLK:= #sROBtoPLC.User.Gripper.DO129_GripperOpen );

   // IF #F_TRIG_Work.Q OR #F_TRIG_Home.Q THEN
   //     "ST10Cylinder".Cy[13].Inout.ManualGoWork := FALSE;
   //     "ST10Cylinder".Cy[13].Inout.ManualGoHome := FALSE;
   // END_IF;

   //<<<<<<<<<<<<<<<<<<<<<<<<<<<<<<<<<<<<<<<<<<<<<<<<<>>>>>>>>>>>>>>>>>>>>>>>>>>>>>>>>>>>>>>>>>>>>>>>>>
   //<<<<<<<<<<<<<<<<<<<<<<<<<<<<<<<<<<<<<<<<  Program End  >>>>>>>>>>>>>>>>>>>>>>>>>>>>>>>>>>>>>>>>>>>
   //<<<<<<<<<<<<<<<<<<<<<<<<<<<<<<<<<<<<<<<<<<<<<<<<<>>>>>>>>>>>>>>>>>>>>>>>>>>>>>>>>>>>>>>>>>>>>>>>>>
END_FUNCTION_BLOCK

FUNCTION_BLOCK "KukaRobot2_Ctrl"   // FB2402, SCL
{ S7_Optimized_Access := 'FALSE' }
// stored: AutoNumber false, SetENOAutomatically false
   VAR_INPUT
      iHWID_In : HW_IO;
      iHWID_Out : HW_IO;
      iSysRun : Bool;
      iAuto : Bool;
      iManual : Bool;
      iSpecial : Bool;
      iE_STOP : Bool;
      iReset : Bool;
      iT1000ms : Bool;
      iTaskMode : USInt;
      iPartType : USInt;
      iSpeedValue : USInt;
      iPGNO : USInt;   // Robot Program number
   END_VAR
   VAR_OUTPUT
      oReady : Bool;
      oStartComplete : Bool;
      oWarning : Bool;
      oError : Bool;
      oErrorCode : Int;
   END_VAR
   VAR_IN_OUT
      ioAutoStart : Bool;
      ioSrartHome : Bool;
      ioStartAutoCycle : Bool;
   END_VAR
   VAR
      sHMI { S7_SetPoint := 'True'} : "KukaRobot_HMI";
      sROBtoPLC : Struct
         Sys { S7_SetPoint := 'True'} : "KukaRobot_SysOutput";   // Robot ---> PLC
         User { S7_SetPoint := 'True'} : "KukaRobot_UserOutput_2";   // Robot ---> PLC
      END_STRUCT;
      sPLCtoROB : Struct
         Sys { S7_SetPoint := 'True'} : "KukaRobot_SysInput";   // PLC ---> Robot
         User { S7_SetPoint := 'True'} : "KukaRobot_UserInput_2";   // PLC ---> Robot
      END_STRUCT;
      sDrivesOnDelay { S7_SetPoint := 'True'} : TON_TIME;
      sStartUpDelay { S7_SetPoint := 'True'} : TON_TIME;
      sRobotReadyToStart : Bool;
      sRobotReadyToRunning : Bool;
      sRobotActComplete : Bool;
      sRobotProgrameChoseOK : Bool;
      sSequence : Int;
      F_TRIG_Work { S7_SetPoint := 'True'} : F_TRIG;
      F_TRIG_Home { S7_SetPoint := 'True'} : F_TRIG;
      ModeValue : Int;
      Tem_ModeValue : Int;
      ModeChange : Bool;
      IEC_Timer_DRIVES_OFF { S7_SetPoint := 'True'} : TON_TIME;
      IEC_Timer_DRIVES_ON { S7_SetPoint := 'True'} : TON_TIME;
   END_VAR
   VAR_TEMP
      tInRwENO : Bool;
      tOutRwENO : Bool;
      tInRwRetVal : Int;
      tOutRwRetVal : Int;
      "tROB-Input" : Array[1..128] of Byte;
      tROB_Output : Array[1..128] of Byte;
   END_VAR
BEGIN
   REGION Description
       (*
       %%%
   VERSION: V1.0
   LANGUAGE: ENGLISH
       %%%
       ** ** ** ** ** ** ** ** ** ** ** ** ** ** ** ** ** ** ** ** ** ** ** ** ** ** ** ** ** ** ** ** ** ** ** ** ** ** ** ** ** ** ** ** ** ** ** ** ** **
       ** ** ** ** ** ** ** ** ** ** ** ** ** ** ** ** ** ** ** ** ** ** ** ** ** ** ** ** ** ** ** ** ** ** ** ** ** ** ** ** ** ** ** ** ** ** ** ** ** **
       * *
       * R (uhlamat) R (obot) I (nterface) *
       * < < Robot Function Block > > *
       * < < Handing Tool > > *
       * - - - - - - - - - - - - - - - - - - - - - - - - - - - - - - - - - - - - - - - - - - *
       * *
       * Customer:   *
       * Roboter Type: Kuka *
       * Software: Siemens TIA V15.1 SP1 *
       * Autor: ChenYi *
       * Company: Ruhlamat Automation Technologies (Suzhou) Co., Ltd *
       * Department: Elec.*
       * Telephone: + 86 (512) 6767 1108 *
       * *
       * Version: 1.0 *
       * Created: 26.05.2020 *
       * Modified: 26.05.2020
   BY: ChenYi *
       * *
       ** ** ** ** ** ** ** ** ** ** ** ** ** ** ** ** ** ** ** ** ** ** ** ** ** ** ** ** ** ** ** ** ** ** ** ** ** ** ** ** ** ** ** ** ** ** ** ** ** **
       ** ** ** ** ** ** ** ** ** ** ** ** ** ** ** ** ** ** ** ** ** ** ** ** ** ** ** ** ** ** ** ** ** ** ** ** ** ** ** ** ** ** ** ** ** ** ** ** ** **
       %%%
    #oErrorCode:
       102:Robot home Failed
       205:Failed to read HW Input data;
       206:Failed to write HW Output data;
       303:Start up TimeOut   

       %%%
       *)
   END_REGION
   //<<<<<<<<<<<<<<<<<<<<<<<<<<<<<<<<<<<<<<<<<<<<<<<<<>>>>>>>>>>>>>>>>>>>>>>>>>>>>>>>>>>>>>>>>>>>>>>>>>
   //<<<<<<<<<<<<<<<<<<<<<<<<<<<<<<<<<<<<<<<<  Program Start  >>>>>>>>>>>>>>>>>>>>>>>>>>>>>>>>>>>>>>>>>
   //<<<<<<<<<<<<<<<<<<<<<<<<<<<<<<<<<<<<<<<<<<<<<<<<<>>>>>>>>>>>>>>>>>>>>>>>>>>>>>>>>>>>>>>>>>>>>>>>>>




   //******************************************
   REGION Bus Input Data Mapping

       #tInRwRetVal := DPRD_DAT(LADDR := #iHWID_In, RECORD => #sROBtoPLC, ENO => #tInRwENO);
       IF NOT #tInRwENO THEN
           GOTO ERROR;
       END_IF;

   END_REGION
   //******************************************
   (*Robot controller remmote control*)

   // I/O Act-Activate interface
   #sPLCtoROB.Sys.SI.I_O_ACT := 1;
   // Move Enable
   //#sPLCtoROB.Sys.SI.MOVE_ENABLE := (#iSysRun AND (((#sROBtoPLC.Sys.SO.T1 OR #sROBtoPLC.Sys.SO.T2) AND #iManual) OR (#iAuto))) AND #iSafePos;
   //#sPLCtoROB.Sys.SI.MOVE_ENABLE := #iSysRun AND (#iManual OR #iAuto) AND #iSafePos;
   IF #sROBtoPLC.Sys.SO.EXT = TRUE THEN
       #sPLCtoROB.Sys.SI.MOVE_ENABLE := #iE_STOP;
   END_IF;
   IF #sROBtoPLC.Sys.SO.T1 = TRUE OR #sROBtoPLC.Sys.SO.T2 = TRUE THEN
       #sPLCtoROB.Sys.SI.MOVE_ENABLE := TRUE;
   END_IF;

   // Drives Off
   #sPLCtoROB.Sys.SI.DRIVES_OFF := NOT #ModeChange;


   IF #iManual
   THEN
       #ModeValue := 1;
   ELSIF #iAuto
   THEN
       #ModeValue := 3;

   END_IF;

   IF #ModeValue <> #Tem_ModeValue
   THEN
       #ModeChange := true;
   ELSE
       #ModeChange := false;
   END_IF;

   IF #IEC_Timer_DRIVES_OFF.Q THEN
       #Tem_ModeValue := #ModeValue;
   END_IF;

   #IEC_Timer_DRIVES_OFF(IN:=#ModeValue <> #Tem_ModeValue,
                         PT:=T#1s);


   //#sPLCtoROB.Sys.SI.DRIVES_OFF := #iSysRun;
   //#sPLCtoROB.Sys.SI.DRIVES_OFF := #iSysRun AND (#iManual OR #iAuto) AND #iSafePos;
   (*Robot controller ready to Start*)
   #sRobotReadyToStart := #iSysRun AND (#iAuto OR #iSpecial) AND
   #sROBtoPLC.Sys.SO.USER_SAF AND #sROBtoPLC.Sys.SO.ALARM_STOP AND
   #sROBtoPLC.Sys.SO.I_O_ACTCONF AND #sROBtoPLC.Sys.SO.ALARM_STOP_INTERN AND
   #sPLCtoROB.Sys.SI.MOVE_ENABLE AND #sPLCtoROB.Sys.SI.DRIVES_OFF
   AND #sROBtoPLC.Sys.SO.EXT;


   REGION Robot Start control
       IF #sRobotReadyToStart THEN
           IF (#sSequence = 0) AND #ioAutoStart AND (#iAuto OR #iSpecial) AND NOT #sRobotActComplete THEN
               #sSequence := 100;
               #ioAutoStart := 0;
               #sRobotActComplete := 0;
               #sRobotProgrameChoseOK := 0;
           END_IF;

           #IEC_Timer_DRIVES_ON(IN := #sSequence=110,
                                 PT := T#100ms);

           CASE #sSequence OF
   (*            100:
                   #sPLCtoROB.Sys.SI.DRIVES_ON := 0;
                   #sSequence := 110;

               110:
                   #sPLCtoROB.Sys.SI.DRIVES_ON := 1;
                   IF #IEC_Timer_DRIVES_ON.Q THEN
                       #sPLCtoROB.Sys.SI.DRIVES_ON := 0;
                       #sSequence := 150;
                   END_IF;
                   *)
               100:  // DrivesOn
                   IF NOT #sROBtoPLC.Sys.SO.RC_RDY1  THEN
                           #sPLCtoROB.Sys.SI.CONF_MESS := 1;
                           #sPLCtoROB.Sys.SI.DRIVES_ON := 0;
                       ELSIF #sROBtoPLC.Sys.SO.RC_RDY1 THEN
                           #sPLCtoROB.Sys.SI.CONF_MESS := 0;
                           #sPLCtoROB.Sys.SI.DRIVES_ON := 1;
                           IF #sDrivesOnDelay.Q AND #sROBtoPLC.Sys.SO.PERI_RDY THEN
                               #sSequence := 200;
                               #sPLCtoROB.Sys.SI.DRIVES_ON := 0;

                           END_IF;
                       END_IF;

                       200:  // ALARM CONF
                       IF #sROBtoPLC.Sys.SO.STOPMESS OR NOT #sROBtoPLC.Sys.SO.RC_RDY1 THEN
                           #sPLCtoROB.Sys.SI.CONF_MESS := 1;
                       ELSE
                           #sPLCtoROB.Sys.SI.CONF_MESS := 0;
                           #sSequence := 300;
                       END_IF;

                       300: // EXT_Start    
                       IF #sROBtoPLC.Sys.SO.PERI_RDY AND NOT #sROBtoPLC.Sys.SO.STOPMESS THEN
                           #sPLCtoROB.Sys.SI.EXT_START := 1;
                           #sSequence := 400;
                       END_IF;

                       400: // EXT_Start Reset  
                       IF #sROBtoPLC.Sys.SO.PRO_ACT THEN
                           #sPLCtoROB.Sys.SI.EXT_START := 0;
                           #sSequence := 500;
                       END_IF;

                       500: // Programe Call
                       IF #sROBtoPLC.Sys.SO.PERI_RDY
                           AND #sROBtoPLC.Sys.SO.PRO_ACT
                           AND #sROBtoPLC.Sys.SO.PGNO_REQ
                           AND #iPGNO <> 0
                           //AND #s_ROBInput.User.User.Home.DI_AutoCycleStart
                           //AND #s_ROBOutput.Sys."SO_$ON_PATH"
                           //AND #s_ROBOutput.Sys."SO_$IN_HOME"
                       THEN

                           #sPLCtoROB.Sys.SI.PGNO_PBIT := #iPGNO;
                           #sPLCtoROB.Sys.SI.PGNO_VALID := 1;
                           #sSequence := 600;
                       END_IF;

                       600: // Programe Call Finish
                       IF #sROBtoPLC.Sys.SO.APPL_RUN THEN
                           #sPLCtoROB.Sys.SI.PGNO_VALID := 0;
                           #sRobotActComplete := 1;
                           #sSequence := 0;
                       END_IF;

           END_CASE;

       ELSE
           #sSequence := 0;
           #sRobotActComplete := 0;
   //        #sPLCtoROB.Sys.SI.DRIVES_ON := 0;////2023/9/1更改
           #sPLCtoROB.Sys.SI.EXT_START := 0;
          // #sPLCtoROB.Sys.SI.CONF_MESS := 0;
           #sPLCtoROB.Sys.SI.PGNO_VALID := 0;
           #sPLCtoROB.Sys.SI.PGNO_PBIT := 0; 
       END_IF;

   (*Robot ready to Running*)
       #sRobotReadyToRunning := #sRobotReadyToStart AND #sROBtoPLC.Sys.SO.PERI_RDY AND #sROBtoPLC.Sys.SO.PRO_ACT AND #sROBtoPLC.Sys.SO.APPL_RUN;


   (*Robot TaskMode,PartType, SpeedValue Set*)
       #sPLCtoROB.User.Public.GI_TaskMode := #iTaskMode;
       #sPLCtoROB.User.Public.GI_PartType := #iPartType;
       #sPLCtoROB.User.Public.GI_SpeedSet := #iSpeedValue;

       // Robot Program calls
       #sPLCtoROB.Sys.SI.PGNO_PARITY := 1;
       //************************************************************
       (*DrivesOn delay*)
       #sDrivesOnDelay(IN := #sPLCtoROB.Sys.SI.DRIVES_ON,
                       PT := T#200ms      // IN: TIME
       );
   (*StartTimeOut delay*)
       #sStartUpDelay(IN := #sSequence <> 0,
                      PT := T#5s        // IN: TIME
       );
       IF #sStartUpDelay.Q THEN
           #sHMI.StartUpTimeOut := 1;
           GOTO ERROR;
       ELSE
           #sHMI.StartUpTimeOut := 0;
       END_IF;

   END_REGION

   //******************************************
   REGION Home
       IF #sRobotReadyToRunning AND #sROBtoPLC.User.Home.DO161_WaitForHomeSeqStart AND NOT #sROBtoPLC.User.Home.DO162_GoHomeFail AND #ioSrartHome THEN
           #sPLCtoROB.User.Home.DI161_HomeSeqStart := 1;
       END_IF;

       IF #sRobotReadyToRunning AND #sROBtoPLC.User.Home.DO163_HomeSeqOK THEN
           #ioSrartHome := 0;
           #sPLCtoROB.User.Home.DI161_HomeSeqStart := 0;
       END_IF;

       IF #sROBtoPLC.User.Home.DO162_GoHomeFail THEN
           GOTO ERROR;
       END_IF;

   END_REGION ;

   REGION Auto Cycle Start

       (*Start Auto Cycle*)
       IF #sRobotReadyToRunning AND #sROBtoPLC.User.Home.DO164_WaitForAutoStart AND #ioStartAutoCycle THEN
           #sPLCtoROB.User.Home.DI162_AutoCycleStart := 1;
       ELSE
           #sPLCtoROB.User.Home.DI162_AutoCycleStart := 0;
       END_IF;

       IF NOT #sROBtoPLC.User.Home.DO164_WaitForAutoStart THEN
           #ioStartAutoCycle := 0;
       END_IF;


   END_REGION ;





   REGION Bus Output Data Mapping

       #tOutRwRetVal := DPWR_DAT(LADDR := #iHWID_Out, RECORD := #sPLCtoROB, ENO => #tOutRwENO);
       IF NOT #tOutRwENO THEN
           GOTO ERROR;
       END_IF;

   END_REGION
   //----------------------------------------------------------------------------------------------------
   REGION Output
       #oReady := #sRobotReadyToRunning;
       #oStartComplete := #sRobotActComplete;


   END_REGION

   REGION HMI Signal
       //SI  
       #sHMI.PGNO_PBIT := #sPLCtoROB.Sys.SI.PGNO_PBIT;
       #sHMI.EXT_START := #sPLCtoROB.Sys.SI.EXT_START;
       #sHMI.MOVE_ENABLE := #sHMI.MOVE_ENABLE;
       #sHMI.CONF_MESS := #sPLCtoROB.Sys.SI.CONF_MESS;
       #sHMI.DRIVES_OFF := NOT #sHMI.DRIVES_OFF;
       #sHMI.DRIVES_ON := #sHMI.DRIVES_ON;
       #sHMI.I_O_ACT := #sHMI.I_O_ACT;
       //UI   
       #sHMI.TaskMode := #sPLCtoROB.User.Public.GI_TaskMode;
       #sHMI.PartType := #sPLCtoROB.User.Public.GI_PartType;
       #sHMI.SpeedSet := #sPLCtoROB.User.Public.GI_SpeedSet;
       #sHMI.HomeSeqStart := #sPLCtoROB.User.Home.DI161_HomeSeqStart;
       #sHMI.AutoCycleStart := #sPLCtoROB.User.Home.DI162_AutoCycleStart;
       //SO   
       #sHMI.RC_RDY1 := #sROBtoPLC.Sys.SO.RC_RDY1;
       #sHMI.ALARM_STOP := NOT #sROBtoPLC.Sys.SO.ALARM_STOP;
       #sHMI.USER_SAF := #sROBtoPLC.Sys.SO.USER_SAF;
       #sHMI.PERI_RDY := #sROBtoPLC.Sys.SO.PERI_RDY;
       #sHMI.ROB_CAL := #sROBtoPLC.Sys.SO.ROB_CAL;
       #sHMI.I_O_ACTCONF := #sROBtoPLC.Sys.SO.I_O_ACTCONF;
       #sHMI.STOPMESS := #sROBtoPLC.Sys.SO.STOPMESS;
       #sHMI.ALARM_STOP_INTERN := NOT #sROBtoPLC.Sys.SO.ALARM_STOP_INTERN;
       #sHMI.PGNO_FBIT_REFL := #sROBtoPLC.Sys.SO.PGNO_FBIT_REFL;
       #sHMI.PRO_ACT := #sROBtoPLC.Sys.SO.PRO_ACT;
       #sHMI.APPL_RUN := #sROBtoPLC.Sys.SO.APPL_RUN;
       #sHMI.PRO_MOVE := #sROBtoPLC.Sys.SO.PRO_MOVE;
       #sHMI.IN_HOME := #sROBtoPLC.Sys.SO.IN_HOME;
       #sHMI.ON_PATH := #sROBtoPLC.Sys.SO.ON_PATH;
       #sHMI.NEAR_POSRET := #sROBtoPLC.Sys.SO.NEAR_POSRET;
       #sHMI.T1 := #sROBtoPLC.Sys.SO.T1;
       #sHMI.T2 := #sROBtoPLC.Sys.SO.T2;
       #sHMI.AUT := #sROBtoPLC.Sys.SO.AUT;
       #sHMI.EXT := #sROBtoPLC.Sys.SO.EXT;
       //UO
       #sHMI.CurrentMode := #sROBtoPLC.User.Public.GO_CurrentMode;
       #sHMI.CurrentPartType := #sROBtoPLC.User.Public.GO_CurrentPartType;
       #sHMI.SpeedActual := #sROBtoPLC.User.Public.GO_SpeedActual;
       #sHMI.ProgramSequence := #sROBtoPLC.User.Public.GO_RobotTaskSequence;
       #sHMI.WaitForHomeSeqStart := #sROBtoPLC.User.Home.DO161_WaitForHomeSeqStart;
       #sHMI.GoHomeFail := #sROBtoPLC.User.Home.DO162_GoHomeFail;
       #sHMI.HomeSeqOK := #sROBtoPLC.User.Home.DO163_HomeSeqOK;
       #sHMI.WaitForAutoCycleStart := #sROBtoPLC.User.Home.DO164_WaitForAutoStart;
       //IO
       #sHMI.iTaskMode := #iTaskMode;
       #sHMI.iPartType := #iPartType;
       #sHMI.iSpeedValue := #iSpeedValue;
       #sHMI.iPGNO := #iPGNO;

       #sHMI.AutoStart := #ioAutoStart;
       #sHMI.SrartHome := #ioSrartHome;
       #sHMI.StartAutoCycle := #ioStartAutoCycle;

       #sHMI.Ready := #oReady;
       #sHMI.StartComplete := #oStartComplete;
       #sHMI.Warning := #oWarning;


   (*Robot working time monitor*)
       IF #iT1000ms AND NOT #sHMI.CountPulse AND #sROBtoPLC.Sys.SO.PERI_RDY THEN
           #sHMI.Seconds := #sHMI.Seconds + 1;
       END_IF;
       #sHMI.CountPulse := #iT1000ms;
       IF #sHMI.Seconds >= 60 THEN
           #sHMI.Minute := #sHMI.Minute + 1;
           #sHMI.Seconds := 0;
       END_IF;
       IF #sHMI.Minute >= 60 THEN
           #sHMI.Hours := #sHMI.Hours + 1;
           #sHMI.Minute := 0;
       END_IF;

   END_REGION

   REGION Error

       IF #iReset AND #oError THEN
           #oError := FALSE;
           #oErrorCode := 0;
       END_IF;

   ERROR:
       ENO := 0;

       IF #sROBtoPLC.User.Home.DO162_GoHomeFail THEN
           #oErrorCode := 102;
       ELSIF #tInRwRetVal <> 0 OR NOT #tInRwENO THEN
           #oError := 1;
           #oErrorCode := 205;
       ELSIF #tOutRwRetVal <> 0 OR NOT #tOutRwENO THEN
           #oError := 1;
           #oErrorCode := 206;
       ELSIF #sStartUpDelay.Q THEN
           #oError := 1;
           #oErrorCode := 303;
       END_IF;



       #sHMI.Error := #oError;
       #sHMI.ErrorCode := #oErrorCode;


   END_REGION

   // IF #sROBtoPLC.User.Gripper.DO129_GripperOpen THEN
   //     "ST10Cylinder".Cy[13].Inout.ManualGoHome := TRUE;
   //     "ST10Cylinder".Cy[13].Inout.ManualGoWork := FALSE;
   // END_IF;

   // IF #sROBtoPLC.User.Gripper.DO130_GripperClose THEN
   //     "ST10Cylinder".Cy[13].Inout.ManualGoWork := TRUE;
   //     "ST10Cylinder".Cy[13].Inout.ManualGoHome := FALSE;
   // END_IF;

   // #F_TRIG_Work(CLK:=#sROBtoPLC.User.Gripper.DO130_GripperClose);

   // #F_TRIG_Home(CLK:= #sROBtoPLC.User.Gripper.DO129_GripperOpen );

   // IF #F_TRIG_Work.Q OR #F_TRIG_Home.Q THEN
   //     "ST10Cylinder".Cy[13].Inout.ManualGoWork := FALSE;
   //     "ST10Cylinder".Cy[13].Inout.ManualGoHome := FALSE;
   // END_IF;

   //<<<<<<<<<<<<<<<<<<<<<<<<<<<<<<<<<<<<<<<<<<<<<<<<<>>>>>>>>>>>>>>>>>>>>>>>>>>>>>>>>>>>>>>>>>>>>>>>>>
   //<<<<<<<<<<<<<<<<<<<<<<<<<<<<<<<<<<<<<<<<  Program End  >>>>>>>>>>>>>>>>>>>>>>>>>>>>>>>>>>>>>>>>>>>
   //<<<<<<<<<<<<<<<<<<<<<<<<<<<<<<<<<<<<<<<<<<<<<<<<<>>>>>>>>>>>>>>>>>>>>>>>>>>>>>>>>>>>>>>>>>>>>>>>>>
END_FUNCTION_BLOCK

FUNCTION_BLOCK "KukaRobot3_Ctrl"   // FB2403, SCL
{ S7_Optimized_Access := 'FALSE' }
// stored: AutoNumber false, SetENOAutomatically false
   VAR_INPUT
      iHWID_In : HW_IO;
      iHWID_Out : HW_IO;
      iSysRun : Bool;
      iAuto : Bool;
      iManual : Bool;
      iSpecial : Bool;
      iE_STOP : Bool;
      iReset : Bool;
      iT1000ms : Bool;
      iTaskMode : USInt;
      iPartType : USInt;
      iSpeedValue : USInt;
      iPGNO : USInt;   // Robot Program number
   END_VAR
   VAR_OUTPUT
      oReady : Bool;
      oStartComplete : Bool;
      oWarning : Bool;
      oError : Bool;
      oErrorCode : Int;
   END_VAR
   VAR_IN_OUT
      ioAutoStart : Bool;
      ioSrartHome : Bool;
      ioStartAutoCycle : Bool;
   END_VAR
   VAR
      sHMI { S7_SetPoint := 'True'} : "KukaRobot_HMI";
      sROBtoPLC : Struct
         Sys { S7_SetPoint := 'True'} : "KukaRobot_SysOutput";   // Robot ---> PLC
         User { S7_SetPoint := 'True'} : "KukaRobot_UserOutput_3";   // Robot ---> PLC
      END_STRUCT;
      sPLCtoROB : Struct
         Sys { S7_SetPoint := 'True'} : "KukaRobot_SysInput";   // PLC ---> Robot
         User { S7_SetPoint := 'True'} : "KukaRobot_UserInput_3";   // PLC ---> Robot
      END_STRUCT;
      sDrivesOnDelay { S7_SetPoint := 'True'} : TON_TIME;
      sStartUpDelay { S7_SetPoint := 'True'} : TON_TIME;
      sRobotReadyToStart : Bool;
      sRobotReadyToRunning : Bool;
      sRobotActComplete : Bool;
      sRobotProgrameChoseOK : Bool;
      sSequence : Int;
      F_TRIG_Work { S7_SetPoint := 'True'} : F_TRIG;
      F_TRIG_Home { S7_SetPoint := 'True'} : F_TRIG;
      ModeValue : Int;
      Tem_ModeValue : Int;
      ModeChange : Bool;
      IEC_Timer_DRIVES_OFF { S7_SetPoint := 'True'} : TON_TIME;
      IEC_Timer_DRIVES_ON { S7_SetPoint := 'True'} : TON_TIME;
   END_VAR
   VAR_TEMP
      tInRwENO : Bool;
      tOutRwENO : Bool;
      tInRwRetVal : Int;
      tOutRwRetVal : Int;
      "tROB-Input" : Array[1..128] of Byte;
      tROB_Output : Array[1..128] of Byte;
   END_VAR
BEGIN
   REGION Description
       (*
       %%%
   VERSION: V1.0
   LANGUAGE: ENGLISH
       %%%
       ** ** ** ** ** ** ** ** ** ** ** ** ** ** ** ** ** ** ** ** ** ** ** ** ** ** ** ** ** ** ** ** ** ** ** ** ** ** ** ** ** ** ** ** ** ** ** ** ** **
       ** ** ** ** ** ** ** ** ** ** ** ** ** ** ** ** ** ** ** ** ** ** ** ** ** ** ** ** ** ** ** ** ** ** ** ** ** ** ** ** ** ** ** ** ** ** ** ** ** **
       * *
       * R (uhlamat) R (obot) I (nterface) *
       * < < Robot Function Block > > *
       * < < Handing Tool > > *
       * - - - - - - - - - - - - - - - - - - - - - - - - - - - - - - - - - - - - - - - - - - *
       * *
       * Customer:   *
       * Roboter Type: Kuka *
       * Software: Siemens TIA V15.1 SP1 *
       * Autor: ChenYi *
       * Company: Ruhlamat Automation Technologies (Suzhou) Co., Ltd *
       * Department: Elec.*
       * Telephone: + 86 (512) 6767 1108 *
       * *
       * Version: 1.0 *
       * Created: 26.05.2020 *
       * Modified: 26.05.2020
   BY: ChenYi *
       * *
       ** ** ** ** ** ** ** ** ** ** ** ** ** ** ** ** ** ** ** ** ** ** ** ** ** ** ** ** ** ** ** ** ** ** ** ** ** ** ** ** ** ** ** ** ** ** ** ** ** **
       ** ** ** ** ** ** ** ** ** ** ** ** ** ** ** ** ** ** ** ** ** ** ** ** ** ** ** ** ** ** ** ** ** ** ** ** ** ** ** ** ** ** ** ** ** ** ** ** ** **
       %%%
    #oErrorCode:
       102:Robot home Failed
       205:Failed to read HW Input data;
       206:Failed to write HW Output data;
       303:Start up TimeOut   

       %%%
       *)
   END_REGION
   //<<<<<<<<<<<<<<<<<<<<<<<<<<<<<<<<<<<<<<<<<<<<<<<<<>>>>>>>>>>>>>>>>>>>>>>>>>>>>>>>>>>>>>>>>>>>>>>>>>
   //<<<<<<<<<<<<<<<<<<<<<<<<<<<<<<<<<<<<<<<<  Program Start  >>>>>>>>>>>>>>>>>>>>>>>>>>>>>>>>>>>>>>>>>
   //<<<<<<<<<<<<<<<<<<<<<<<<<<<<<<<<<<<<<<<<<<<<<<<<<>>>>>>>>>>>>>>>>>>>>>>>>>>>>>>>>>>>>>>>>>>>>>>>>>




   //******************************************
   REGION Bus Input Data Mapping

       #tInRwRetVal := DPRD_DAT(LADDR := #iHWID_In, RECORD => #sROBtoPLC, ENO => #tInRwENO);
       IF NOT #tInRwENO THEN
           GOTO ERROR;
       END_IF;

   END_REGION
   //******************************************
   (*Robot controller remmote control*)

   // I/O Act-Activate interface
   #sPLCtoROB.Sys.SI.I_O_ACT := 1;
   // Move Enable
   //#sPLCtoROB.Sys.SI.MOVE_ENABLE := (#iSysRun AND (((#sROBtoPLC.Sys.SO.T1 OR #sROBtoPLC.Sys.SO.T2) AND #iManual) OR (#iAuto))) AND #iSafePos;
   //#sPLCtoROB.Sys.SI.MOVE_ENABLE := #iSysRun AND (#iManual OR #iAuto) AND #iSafePos;
   IF #sROBtoPLC.Sys.SO.EXT = TRUE THEN
       #sPLCtoROB.Sys.SI.MOVE_ENABLE := #iE_STOP;
   END_IF;
   IF #sROBtoPLC.Sys.SO.T1 = TRUE OR #sROBtoPLC.Sys.SO.T2 = TRUE THEN
       #sPLCtoROB.Sys.SI.MOVE_ENABLE := TRUE;
   END_IF;
   // Drives Off
   #sPLCtoROB.Sys.SI.DRIVES_OFF := NOT #ModeChange;


   IF #iManual
   THEN
       #ModeValue := 1;
   ELSIF #iAuto
   THEN
       #ModeValue := 3;

   END_IF;

   IF #ModeValue <> #Tem_ModeValue
   THEN
       #ModeChange := true;
   ELSE
       #ModeChange := false;
   END_IF;

   IF #IEC_Timer_DRIVES_OFF.Q THEN
       #Tem_ModeValue := #ModeValue;
   END_IF;

   #IEC_Timer_DRIVES_OFF(IN:=#ModeValue <> #Tem_ModeValue,
                         PT:=T#1s);


   //#sPLCtoROB.Sys.SI.DRIVES_OFF := #iSysRun;
   //#sPLCtoROB.Sys.SI.DRIVES_OFF := #iSysRun AND (#iManual OR #iAuto) AND #iSafePos;
   (*Robot controller ready to Start*)
   #sRobotReadyToStart := #iSysRun AND (#iAuto OR #iSpecial) AND
   #sROBtoPLC.Sys.SO.USER_SAF AND #sROBtoPLC.Sys.SO.ALARM_STOP AND
   #sROBtoPLC.Sys.SO.I_O_ACTCONF AND #sROBtoPLC.Sys.SO.ALARM_STOP_INTERN AND
   #sPLCtoROB.Sys.SI.MOVE_ENABLE AND #sPLCtoROB.Sys.SI.DRIVES_OFF
   AND #sROBtoPLC.Sys.SO.EXT;


   REGION Robot Start control
       IF #sRobotReadyToStart THEN
           IF (#sSequence = 0) AND #ioAutoStart AND (#iAuto OR #iSpecial) AND NOT #sRobotActComplete THEN
               #sSequence := 100;
               #ioAutoStart := 0;
               #sRobotActComplete := 0;
               #sRobotProgrameChoseOK := 0;
           END_IF;

           #IEC_Timer_DRIVES_ON(IN := #sSequence=110,
                                 PT := T#100ms);

           CASE #sSequence OF
   (*            100:
                   #sPLCtoROB.Sys.SI.DRIVES_ON := 0;
                   #sSequence := 110;

               110:
                   #sPLCtoROB.Sys.SI.DRIVES_ON := 1;
                   IF #IEC_Timer_DRIVES_ON.Q THEN
                       #sPLCtoROB.Sys.SI.DRIVES_ON := 0;
                       #sSequence := 150;
                   END_IF;
                   *)
               100:  // DrivesOn
                   IF NOT #sROBtoPLC.Sys.SO.RC_RDY1  THEN
                           #sPLCtoROB.Sys.SI.CONF_MESS := 1;
                           #sPLCtoROB.Sys.SI.DRIVES_ON := 0;
                       ELSIF #sROBtoPLC.Sys.SO.RC_RDY1 THEN
                           #sPLCtoROB.Sys.SI.CONF_MESS := 0;
                           #sPLCtoROB.Sys.SI.DRIVES_ON := 1;
                           IF #sDrivesOnDelay.Q AND #sROBtoPLC.Sys.SO.PERI_RDY THEN
                               #sSequence := 200;
                               #sPLCtoROB.Sys.SI.DRIVES_ON := 0;

                           END_IF;
                       END_IF;

                       200:  // ALARM CONF
                       IF #sROBtoPLC.Sys.SO.STOPMESS OR NOT #sROBtoPLC.Sys.SO.RC_RDY1 THEN
                           #sPLCtoROB.Sys.SI.CONF_MESS := 1;
                       ELSE
                           #sPLCtoROB.Sys.SI.CONF_MESS := 0;
                           #sSequence := 300;
                       END_IF;

                       300: // EXT_Start    
                       IF #sROBtoPLC.Sys.SO.PERI_RDY AND NOT #sROBtoPLC.Sys.SO.STOPMESS THEN
                           #sPLCtoROB.Sys.SI.EXT_START := 1;
                           #sSequence := 400;
                       END_IF;

                       400: // EXT_Start Reset  
                       IF #sROBtoPLC.Sys.SO.PRO_ACT THEN
                           #sPLCtoROB.Sys.SI.EXT_START := 0;
                           #sSequence := 500;
                       END_IF;

                       500: // Programe Call
                       IF #sROBtoPLC.Sys.SO.PERI_RDY
                           AND #sROBtoPLC.Sys.SO.PRO_ACT
                           AND #sROBtoPLC.Sys.SO.PGNO_REQ
                           AND #iPGNO <> 0
                           //AND #s_ROBInput.User.User.Home.DI_AutoCycleStart
                           //AND #s_ROBOutput.Sys."SO_$ON_PATH"
                           //AND #s_ROBOutput.Sys."SO_$IN_HOME"
                       THEN

                           #sPLCtoROB.Sys.SI.PGNO_PBIT := #iPGNO;
                           #sPLCtoROB.Sys.SI.PGNO_VALID := 1;
                           #sSequence := 600;
                       END_IF;

                       600: // Programe Call Finish
                       IF #sROBtoPLC.Sys.SO.APPL_RUN THEN
                           #sPLCtoROB.Sys.SI.PGNO_VALID := 0;
                           #sRobotActComplete := 1;
                           #sSequence := 0;
                       END_IF;

           END_CASE;

       ELSE
           #sSequence := 0;
           #sRobotActComplete := 0;
   //        #sPLCtoROB.Sys.SI.DRIVES_ON := 0;////2023/9/1更改
           #sPLCtoROB.Sys.SI.EXT_START := 0;
          // #sPLCtoROB.Sys.SI.CONF_MESS := 0;
           #sPLCtoROB.Sys.SI.PGNO_VALID := 0;
           #sPLCtoROB.Sys.SI.PGNO_PBIT := 0; 
       END_IF;

   (*Robot ready to Running*)
       #sRobotReadyToRunning := #sRobotReadyToStart AND #sROBtoPLC.Sys.SO.PERI_RDY AND #sROBtoPLC.Sys.SO.PRO_ACT AND #sROBtoPLC.Sys.SO.APPL_RUN;


   (*Robot TaskMode,PartType, SpeedValue Set*)
       #sPLCtoROB.User.Public.GI_TaskMode := #iTaskMode;
       #sPLCtoROB.User.Public.GI_PartType := #iPartType;
       #sPLCtoROB.User.Public.GI_SpeedSet := #iSpeedValue;

       // Robot Program calls
       #sPLCtoROB.Sys.SI.PGNO_PARITY := 1;
       //************************************************************
       (*DrivesOn delay*)
       #sDrivesOnDelay(IN := #sPLCtoROB.Sys.SI.DRIVES_ON,
                       PT := T#200ms      // IN: TIME
       );
   (*StartTimeOut delay*)
       #sStartUpDelay(IN := #sSequence <> 0,
                      PT := T#5s        // IN: TIME
       );
       IF #sStartUpDelay.Q THEN
           #sHMI.StartUpTimeOut := 1;
           GOTO ERROR;
       ELSE
           #sHMI.StartUpTimeOut := 0;
       END_IF;

   END_REGION

   //******************************************
   REGION Home
       IF #sRobotReadyToRunning AND #sROBtoPLC.User.Home.DO161_WaitForHomeSeqStart AND NOT #sROBtoPLC.User.Home.DO162_GoHomeFail AND #ioSrartHome THEN
           #sPLCtoROB.User.Home.DI161_HomeSeqStart := 1;
       END_IF;

       IF #sRobotReadyToRunning AND #sROBtoPLC.User.Home.DO163_HomeSeqOK THEN
           #ioSrartHome := 0;
           #sPLCtoROB.User.Home.DI161_HomeSeqStart := 0;
       END_IF;

       IF #sROBtoPLC.User.Home.DO162_GoHomeFail THEN
           GOTO ERROR;
       END_IF;

   END_REGION ;

   REGION Auto Cycle Start

       (*Start Auto Cycle*)
       IF #sRobotReadyToRunning AND #sROBtoPLC.User.Home.DO164_WaitForAutoStart AND #ioStartAutoCycle THEN
           #sPLCtoROB.User.Home.DI162_AutoCycleStart := 1;
       ELSE
           #sPLCtoROB.User.Home.DI162_AutoCycleStart := 0;
       END_IF;

       IF NOT #sROBtoPLC.User.Home.DO164_WaitForAutoStart THEN
           #ioStartAutoCycle := 0;
       END_IF;


   END_REGION ;





   REGION Bus Output Data Mapping

       #tOutRwRetVal := DPWR_DAT(LADDR := #iHWID_Out, RECORD := #sPLCtoROB, ENO => #tOutRwENO);
       IF NOT #tOutRwENO THEN
           GOTO ERROR;
       END_IF;

   END_REGION
   //----------------------------------------------------------------------------------------------------
   REGION Output
       #oReady := #sRobotReadyToRunning;
       #oStartComplete := #sRobotActComplete;


   END_REGION

   REGION HMI Signal
       //SI  
       #sHMI.PGNO_PBIT := #sPLCtoROB.Sys.SI.PGNO_PBIT;
       #sHMI.EXT_START := #sPLCtoROB.Sys.SI.EXT_START;
       #sHMI.MOVE_ENABLE := #sHMI.MOVE_ENABLE;
       #sHMI.CONF_MESS := #sPLCtoROB.Sys.SI.CONF_MESS;
       #sHMI.DRIVES_OFF := NOT #sHMI.DRIVES_OFF;
       #sHMI.DRIVES_ON := #sHMI.DRIVES_ON;
       #sHMI.I_O_ACT := #sHMI.I_O_ACT;
       //UI   
       #sHMI.TaskMode := #sPLCtoROB.User.Public.GI_TaskMode;
       #sHMI.PartType := #sPLCtoROB.User.Public.GI_PartType;
       #sHMI.SpeedSet := #sPLCtoROB.User.Public.GI_SpeedSet;
       #sHMI.HomeSeqStart := #sPLCtoROB.User.Home.DI161_HomeSeqStart;
       #sHMI.AutoCycleStart := #sPLCtoROB.User.Home.DI162_AutoCycleStart;
       //SO   
       #sHMI.RC_RDY1 := #sROBtoPLC.Sys.SO.RC_RDY1;
       #sHMI.ALARM_STOP := NOT #sROBtoPLC.Sys.SO.ALARM_STOP;
       #sHMI.USER_SAF := #sROBtoPLC.Sys.SO.USER_SAF;
       #sHMI.PERI_RDY := #sROBtoPLC.Sys.SO.PERI_RDY;
       #sHMI.ROB_CAL := #sROBtoPLC.Sys.SO.ROB_CAL;
       #sHMI.I_O_ACTCONF := #sROBtoPLC.Sys.SO.I_O_ACTCONF;
       #sHMI.STOPMESS := #sROBtoPLC.Sys.SO.STOPMESS;
       #sHMI.ALARM_STOP_INTERN := NOT #sROBtoPLC.Sys.SO.ALARM_STOP_INTERN;
       #sHMI.PGNO_FBIT_REFL := #sROBtoPLC.Sys.SO.PGNO_FBIT_REFL;
       #sHMI.PRO_ACT := #sROBtoPLC.Sys.SO.PRO_ACT;
       #sHMI.APPL_RUN := #sROBtoPLC.Sys.SO.APPL_RUN;
       #sHMI.PRO_MOVE := #sROBtoPLC.Sys.SO.PRO_MOVE;
       #sHMI.IN_HOME := #sROBtoPLC.Sys.SO.IN_HOME;
       #sHMI.ON_PATH := #sROBtoPLC.Sys.SO.ON_PATH;
       #sHMI.NEAR_POSRET := #sROBtoPLC.Sys.SO.NEAR_POSRET;
       #sHMI.T1 := #sROBtoPLC.Sys.SO.T1;
       #sHMI.T2 := #sROBtoPLC.Sys.SO.T2;
       #sHMI.AUT := #sROBtoPLC.Sys.SO.AUT;
       #sHMI.EXT := #sROBtoPLC.Sys.SO.EXT;
       //UO
       #sHMI.CurrentMode := #sROBtoPLC.User.Public.GO_CurrentMode;
       #sHMI.CurrentPartType := #sROBtoPLC.User.Public.GO_CurrentPartType;
       #sHMI.SpeedActual := #sROBtoPLC.User.Public.GO_SpeedActual;
       #sHMI.ProgramSequence := #sROBtoPLC.User.Public.GO_RobotTaskSequence;
       #sHMI.WaitForHomeSeqStart := #sROBtoPLC.User.Home.DO161_WaitForHomeSeqStart;
       #sHMI.GoHomeFail := #sROBtoPLC.User.Home.DO162_GoHomeFail;
       #sHMI.HomeSeqOK := #sROBtoPLC.User.Home.DO163_HomeSeqOK;
       #sHMI.WaitForAutoCycleStart := #sROBtoPLC.User.Home.DO164_WaitForAutoStart;
       //IO
       #sHMI.iTaskMode := #iTaskMode;
       #sHMI.iPartType := #iPartType;
       #sHMI.iSpeedValue := #iSpeedValue;
       #sHMI.iPGNO := #iPGNO;

       #sHMI.AutoStart := #ioAutoStart;
       #sHMI.SrartHome := #ioSrartHome;
       #sHMI.StartAutoCycle := #ioStartAutoCycle;

       #sHMI.Ready := #oReady;
       #sHMI.StartComplete := #oStartComplete;
       #sHMI.Warning := #oWarning;


   (*Robot working time monitor*)
       IF #iT1000ms AND NOT #sHMI.CountPulse AND #sROBtoPLC.Sys.SO.PERI_RDY THEN
           #sHMI.Seconds := #sHMI.Seconds + 1;
       END_IF;
       #sHMI.CountPulse := #iT1000ms;
       IF #sHMI.Seconds >= 60 THEN
           #sHMI.Minute := #sHMI.Minute + 1;
           #sHMI.Seconds := 0;
       END_IF;
       IF #sHMI.Minute >= 60 THEN
           #sHMI.Hours := #sHMI.Hours + 1;
           #sHMI.Minute := 0;
       END_IF;

   END_REGION

   REGION Error

       IF #iReset AND #oError THEN
           #oError := FALSE;
           #oErrorCode := 0;
       END_IF;

   ERROR:
       ENO := 0;

       IF #sROBtoPLC.User.Home.DO162_GoHomeFail THEN
           #oErrorCode := 102;
       ELSIF #tInRwRetVal <> 0 OR NOT #tInRwENO THEN
           #oError := 1;
           #oErrorCode := 205;
       ELSIF #tOutRwRetVal <> 0 OR NOT #tOutRwENO THEN
           #oError := 1;
           #oErrorCode := 206;
       ELSIF #sStartUpDelay.Q THEN
           #oError := 1;
           #oErrorCode := 303;
       END_IF;



       #sHMI.Error := #oError;
       #sHMI.ErrorCode := #oErrorCode;


   END_REGION

   // IF #sROBtoPLC.User.Gripper.DO129_GripperOpen THEN
   //     "ST10Cylinder".Cy[13].Inout.ManualGoHome := TRUE;
   //     "ST10Cylinder".Cy[13].Inout.ManualGoWork := FALSE;
   // END_IF;

   // IF #sROBtoPLC.User.Gripper.DO130_GripperClose THEN
   //     "ST10Cylinder".Cy[13].Inout.ManualGoWork := TRUE;
   //     "ST10Cylinder".Cy[13].Inout.ManualGoHome := FALSE;
   // END_IF;

   // #F_TRIG_Work(CLK:=#sROBtoPLC.User.Gripper.DO130_GripperClose);

   // #F_TRIG_Home(CLK:= #sROBtoPLC.User.Gripper.DO129_GripperOpen );

   // IF #F_TRIG_Work.Q OR #F_TRIG_Home.Q THEN
   //     "ST10Cylinder".Cy[13].Inout.ManualGoWork := FALSE;
   //     "ST10Cylinder".Cy[13].Inout.ManualGoHome := FALSE;
   // END_IF;

   //<<<<<<<<<<<<<<<<<<<<<<<<<<<<<<<<<<<<<<<<<<<<<<<<<>>>>>>>>>>>>>>>>>>>>>>>>>>>>>>>>>>>>>>>>>>>>>>>>>
   //<<<<<<<<<<<<<<<<<<<<<<<<<<<<<<<<<<<<<<<<  Program End  >>>>>>>>>>>>>>>>>>>>>>>>>>>>>>>>>>>>>>>>>>>
   //<<<<<<<<<<<<<<<<<<<<<<<<<<<<<<<<<<<<<<<<<<<<<<<<<>>>>>>>>>>>>>>>>>>>>>>>>>>>>>>>>>>>>>>>>>>>>>>>>>
END_FUNCTION_BLOCK

FUNCTION "SR1000" : Void   // FC1800, LAD
{ S7_Optimized_Access := 'TRUE' }
// stored: AutoNumber false, SetENOAutomatically false
BEGIN

REGION Network 1: 801A1
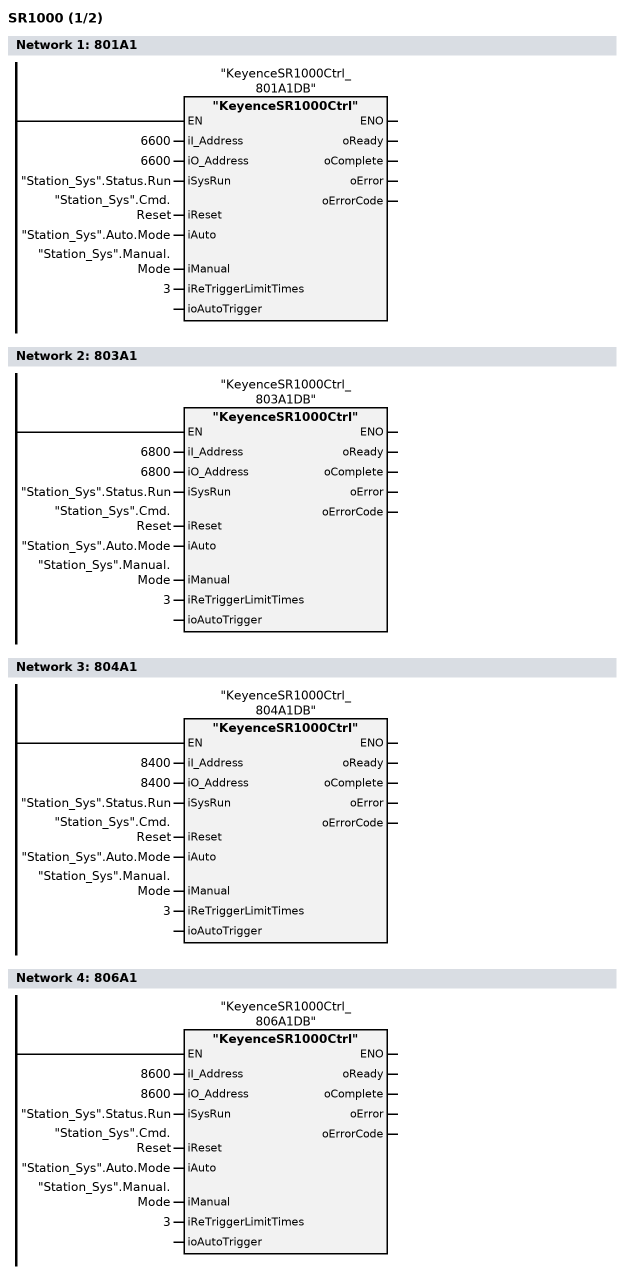
   RUNG wire#powerrail
      "KeyenceSR1000Ctrl_801A1DB"(iI_Address := 6600, iO_Address := 6600, iSysRun := "Station_Sys".Status.Run, iReset := "Station_Sys".Cmd.Reset, iAuto := "Station_Sys".Auto.Mode, iManual := "Station_Sys".Manual.Mode, iReTriggerLimitTimes := 3, ioAutoTrigger :=, oReady =>, oComplete =>, oError =>, oErrorCode =>)
   END_RUNG
   // the same network as SCL:
   "KeyenceSR1000Ctrl_801A1DB"(iI_Address := 6600,   // "KeyenceSR1000Ctrl"
                           iO_Address := 6600,
                           iSysRun := "Station_Sys".Status.Run,
                           iReset := "Station_Sys".Cmd.Reset,
                           iAuto := "Station_Sys".Auto.Mode,
                           iManual := "Station_Sys".Manual.Mode,
                           iReTriggerLimitTimes := 3);
END_REGION

REGION Network 2: 803A1
   RUNG wire#powerrail
      "KeyenceSR1000Ctrl_803A1DB"(iI_Address := 6800, iO_Address := 6800, iSysRun := "Station_Sys".Status.Run, iReset := "Station_Sys".Cmd.Reset, iAuto := "Station_Sys".Auto.Mode, iManual := "Station_Sys".Manual.Mode, iReTriggerLimitTimes := 3, ioAutoTrigger :=, oReady =>, oComplete =>, oError =>, oErrorCode =>)
   END_RUNG
   // the same network as SCL:
   "KeyenceSR1000Ctrl_803A1DB"(iI_Address := 6800,   // "KeyenceSR1000Ctrl"
                           iO_Address := 6800,
                           iSysRun := "Station_Sys".Status.Run,
                           iReset := "Station_Sys".Cmd.Reset,
                           iAuto := "Station_Sys".Auto.Mode,
                           iManual := "Station_Sys".Manual.Mode,
                           iReTriggerLimitTimes := 3);
END_REGION

REGION Network 3: 804A1
   RUNG wire#powerrail
      "KeyenceSR1000Ctrl_804A1DB"(iI_Address := 8400, iO_Address := 8400, iSysRun := "Station_Sys".Status.Run, iReset := "Station_Sys".Cmd.Reset, iAuto := "Station_Sys".Auto.Mode, iManual := "Station_Sys".Manual.Mode, iReTriggerLimitTimes := 3, ioAutoTrigger :=, oReady =>, oComplete =>, oError =>, oErrorCode =>)
   END_RUNG
   // the same network as SCL:
   "KeyenceSR1000Ctrl_804A1DB"(iI_Address := 8400,   // "KeyenceSR1000Ctrl"
                           iO_Address := 8400,
                           iSysRun := "Station_Sys".Status.Run,
                           iReset := "Station_Sys".Cmd.Reset,
                           iAuto := "Station_Sys".Auto.Mode,
                           iManual := "Station_Sys".Manual.Mode,
                           iReTriggerLimitTimes := 3);
END_REGION

REGION Network 4: 806A1
   RUNG wire#powerrail
      "KeyenceSR1000Ctrl_806A1DB"(iI_Address := 8600, iO_Address := 8600, iSysRun := "Station_Sys".Status.Run, iReset := "Station_Sys".Cmd.Reset, iAuto := "Station_Sys".Auto.Mode, iManual := "Station_Sys".Manual.Mode, iReTriggerLimitTimes := 3, ioAutoTrigger :=, oReady =>, oComplete =>, oError =>, oErrorCode =>)
   END_RUNG
   // the same network as SCL:
   "KeyenceSR1000Ctrl_806A1DB"(iI_Address := 8600,   // "KeyenceSR1000Ctrl"
                           iO_Address := 8600,
                           iSysRun := "Station_Sys".Status.Run,
                           iReset := "Station_Sys".Cmd.Reset,
                           iAuto := "Station_Sys".Auto.Mode,
                           iManual := "Station_Sys".Manual.Mode,
                           iReTriggerLimitTimes := 3);
END_REGION

REGION Network 5: 800A1
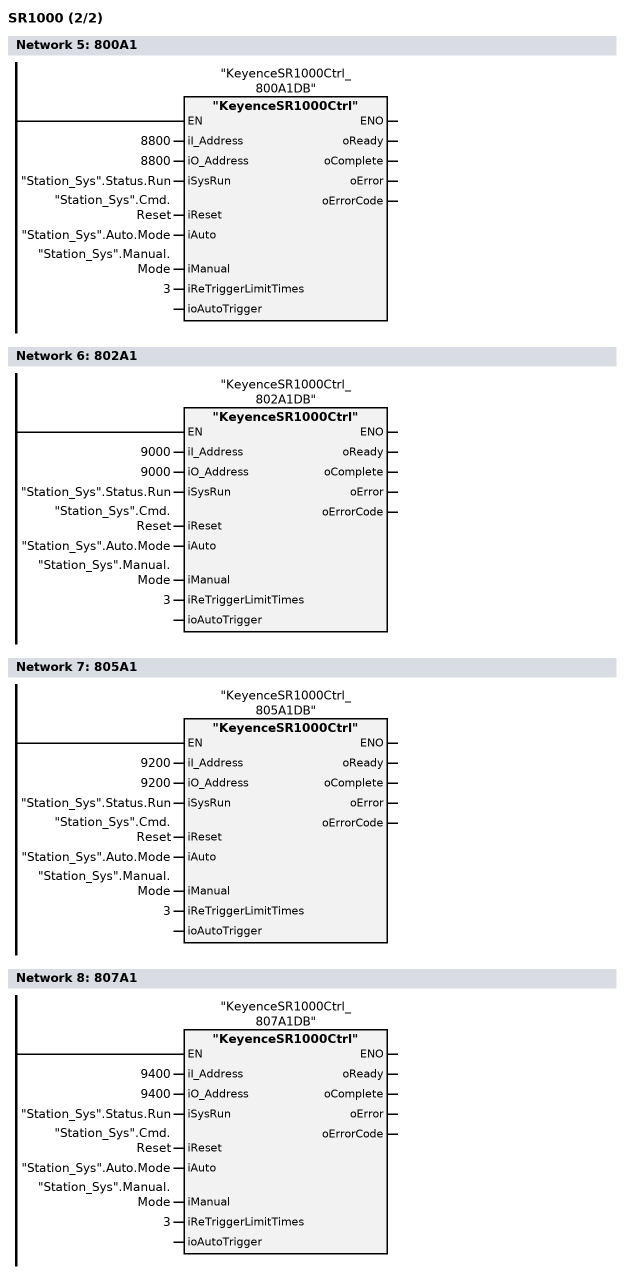
   RUNG wire#powerrail
      "KeyenceSR1000Ctrl_800A1DB"(iI_Address := 8800, iO_Address := 8800, iSysRun := "Station_Sys".Status.Run, iReset := "Station_Sys".Cmd.Reset, iAuto := "Station_Sys".Auto.Mode, iManual := "Station_Sys".Manual.Mode, iReTriggerLimitTimes := 3, ioAutoTrigger :=, oReady =>, oComplete =>, oError =>, oErrorCode =>)
   END_RUNG
   // the same network as SCL:
   "KeyenceSR1000Ctrl_800A1DB"(iI_Address := 8800,   // "KeyenceSR1000Ctrl"
                           iO_Address := 8800,
                           iSysRun := "Station_Sys".Status.Run,
                           iReset := "Station_Sys".Cmd.Reset,
                           iAuto := "Station_Sys".Auto.Mode,
                           iManual := "Station_Sys".Manual.Mode,
                           iReTriggerLimitTimes := 3);
END_REGION

REGION Network 6: 802A1
   RUNG wire#powerrail
      "KeyenceSR1000Ctrl_802A1DB"(iI_Address := 9000, iO_Address := 9000, iSysRun := "Station_Sys".Status.Run, iReset := "Station_Sys".Cmd.Reset, iAuto := "Station_Sys".Auto.Mode, iManual := "Station_Sys".Manual.Mode, iReTriggerLimitTimes := 3, ioAutoTrigger :=, oReady =>, oComplete =>, oError =>, oErrorCode =>)
   END_RUNG
   // the same network as SCL:
   "KeyenceSR1000Ctrl_802A1DB"(iI_Address := 9000,   // "KeyenceSR1000Ctrl"
                           iO_Address := 9000,
                           iSysRun := "Station_Sys".Status.Run,
                           iReset := "Station_Sys".Cmd.Reset,
                           iAuto := "Station_Sys".Auto.Mode,
                           iManual := "Station_Sys".Manual.Mode,
                           iReTriggerLimitTimes := 3);
END_REGION

REGION Network 7: 805A1
   RUNG wire#powerrail
      "KeyenceSR1000Ctrl_805A1DB"(iI_Address := 9200, iO_Address := 9200, iSysRun := "Station_Sys".Status.Run, iReset := "Station_Sys".Cmd.Reset, iAuto := "Station_Sys".Auto.Mode, iManual := "Station_Sys".Manual.Mode, iReTriggerLimitTimes := 3, ioAutoTrigger :=, oReady =>, oComplete =>, oError =>, oErrorCode =>)
   END_RUNG
   // the same network as SCL:
   "KeyenceSR1000Ctrl_805A1DB"(iI_Address := 9200,   // "KeyenceSR1000Ctrl"
                           iO_Address := 9200,
                           iSysRun := "Station_Sys".Status.Run,
                           iReset := "Station_Sys".Cmd.Reset,
                           iAuto := "Station_Sys".Auto.Mode,
                           iManual := "Station_Sys".Manual.Mode,
                           iReTriggerLimitTimes := 3);
END_REGION

REGION Network 8: 807A1
   RUNG wire#powerrail
      "KeyenceSR1000Ctrl_807A1DB"(iI_Address := 9400, iO_Address := 9400, iSysRun := "Station_Sys".Status.Run, iReset := "Station_Sys".Cmd.Reset, iAuto := "Station_Sys".Auto.Mode, iManual := "Station_Sys".Manual.Mode, iReTriggerLimitTimes := 3, ioAutoTrigger :=, oReady =>, oComplete =>, oError =>, oErrorCode =>)
   END_RUNG
   // the same network as SCL:
   "KeyenceSR1000Ctrl_807A1DB"(iI_Address := 9400,   // "KeyenceSR1000Ctrl"
                           iO_Address := 9400,
                           iSysRun := "Station_Sys".Status.Run,
                           iReset := "Station_Sys".Cmd.Reset,
                           iAuto := "Station_Sys".Auto.Mode,
                           iManual := "Station_Sys".Manual.Mode,
                           iReTriggerLimitTimes := 3);
END_REGION
END_FUNCTION

FUNCTION_BLOCK "KeyenceSR1000Ctrl"   // FB1800, SCL
{ S7_Optimized_Access := 'FALSE' }
// stored: AutoNumber false, SetENOAutomatically false
   VAR_INPUT
      iI_Address { ExternalAccessible := 'False'; ExternalVisible := 'False'; ExternalWritable := 'False'} : Int;   // hardware first input address
      iO_Address : Int;   // hardware first Output address
      iSysRun : Bool;
      iReset : Bool;
      iAuto : Bool;
      iManual : Bool;
      iReTriggerLimitTimes : USInt := 3;
   END_VAR
   VAR_OUTPUT
      oReady : Bool;
      oComplete : Bool;
      oError : Bool;
      oErrorCode : UInt;
   END_VAR
   VAR_IN_OUT
      ioAutoTrigger : Bool;
   END_VAR
   VAR
      sHMI { S7_SetPoint := 'True'} : "RCS_KeyenceSR1000_HMI1";
      sCtrl : Struct
         Sequence : Int;
      END_STRUCT;
      sCurrentCode : String[128];
      sAtCurrentCode AT sCurrentCode : Array[-1..128] of Byte;
      sInData { S7_SetPoint := 'True'} : "RCS_KeyenceSR1000_Input1";
      sOutData { S7_SetPoint := 'True'} : "RCS_KeyenceSR1000_Output1";
      sAutoOld : Bool;
      sManualOld : Bool;
      sBusyTimeOut : Bool;
      sRunTimer { S7_SetPoint := 'True'} : TON_TIME;
      sBusyTimer { S7_SetPoint := 'True'} : TON_TIME;
      sFindCurrentPos { S7_SetPoint := 'True'} : Int;
   END_VAR
   VAR_TEMP
      tAny : Any;
      tAnyParameters AT tAny : Struct
         SyntaxID : Byte;
         DataType : Byte;
         RepetitionFactor : Int;
         DB_Number : Word;
         MemoryAreaAddress : DWord;
      END_STRUCT;
      tOffset : Int;
      tEmpty : DWord;
      tIndex : Int;
      tRetVal : Int;
   END_VAR
BEGIN
   REGION Description
   (*
   KEYENCE SR-1000 Reader Function Block
   ruhlamat Automation Technologies(Suzhou) Co.,Ltd
   Copyright(c) 2020.All rights reserved.
   -------------------------------------------------------------------------------------------
   NAME OF FUNCTION BLOCK:"SR-1000Ctrl"
   NUMBER OF FUNCTION BLOCK: FB4021
   FAMILY:ruhlamat PSL
   VERSION:V1.0
   AUTHOR:Qianfeng.Yang
   LAST CHANGE:06.05.2021 (DB)
   -------------------------------------------------------------------------------------------
   Date Name Activity
   06.29.2020 Created by Qianfeng.Yang(V1.0)
   -------------------------------------------------------------------------------------------
   *)
   (*
   Trigger method: Level trigger. Handshaking: Disabled

   When reading is successful#################################################
   1 "Read request" is set to ON (1).
   2 When "Read request" is set to ON (1), the SR-1000 Series starts reading,and then "TRG BUSY" is set to ON (1).
   3 When the code is read, its data is written into "Read Data." "TRG BUSY" is set to OFF (0), and "Read Complete" is set to ON (1).
   4 "Read request" is set to OFF (0).
   5 It is confirmed that "Read Complete" is ON (1), and then "Read Complete Clear" is set to ON (1).
   6 When "Read Complete Clear" is set to ON (1), "Read Complete" is set to OFF (0).
   7 It is confirmed that "Read Complete" is OFF (0), and then "Read Complete Clear" is set to OFF (0).

   When reading fails##########################################################
   1 "Read request" is set to ON (1).
   2 When "Read request" is set to ON (1), the SR-1000 Series starts reading,and then "TRG BUSY" is set to ON (1).
   3 "Read request" is set to OFF (0).
   4 The code could not be read, so "ERROR" is written to "Result Data." "201" is written to "Read Result Code." "TRG BUSY" is set to OFF (0), and "Read Complete" is set to ON (1).
   5 It is confirmed that "Read Complete" is ON (1), and then "Read Complete Clear" is set to ON (1).
   6 When "Read Complete Clear" is set to ON (1), "Read Complete" and "Read Failure" are set to OFF (0).
   7 It is confirmed that "Read Complete" is OFF (0), and then "Read Complete Clear" is set to OFF (0).
   *)
   (*
   Error code List
     0=No error / (Reading success/operation succes)
   201=Reading error
   202=Comparison error / (The read code does not match the preset data)
   210=Tuning failure(Symbol unclear) / (The code could not be found within the field of)
   213=Tuning failure(Aborted) / (Tuning was aborted midwayview while tuning.)
   120=Control instruction receptionerror / (Another operation instruction was received during operation. (Operation instruction is notcompleted.)
   102=Bank No. error / (The bank number specification is invalid(other than 1 to 16))
   220=Preset data error / (Preset data specification is invalid.(Specified size is outside the range.))
   230=PROFINET data update error / (Shortage of specified size (Result data and present data size is beyond the limit.))

   FB ERROR
   1205=Failed to read HW Input data
   1206=Failed to write HW Output data
   1303=PG Running Timeout
   *)
   END_REGION

   (*Begin*)
   (*Read Data from KEYENCE SR-1000 TO PLC memory*)
   REGION Read inputs    
       #tAnyParameters.SyntaxID := 16#10;
       #tAnyParameters.DataType := 16#02;//Data type:Byte
       #tOffset := #iI_Address;
       #tAnyParameters.RepetitionFactor := 1;
       #tAnyParameters.DB_Number := 16#0;
       #tAnyParameters.MemoryAreaAddress := 16#8100_0000 OR (SHL(IN := INT_TO_DWORD(#tOffset), N := 3)); //B#16#81 Input Area
       IF BLKMOV(SRCBLK := #tAny, DSTBLK => #sInData.HandshakeAndGeneralErrorStatus) <> 0 THEN
           #sHMI.Status.Error := 1;
           #sHMI.Status.ErrorCode := 1205;
           GOTO Error;
       END_IF;
       #tOffset += #tAnyParameters.RepetitionFactor;
       #tAnyParameters.RepetitionFactor := 1;
       #tAnyParameters.MemoryAreaAddress := 16#8100_0000 OR (SHL(IN := INT_TO_DWORD(#tOffset), N := 3));
       IF BLKMOV(SRCBLK := #tAny, DSTBLK => #sInData.BusyStatus) <> 0 THEN
           #sHMI.Status.Error := 1;
           #sHMI.Status.ErrorCode := 1205;
           GOTO Error;
       END_IF;
       #tOffset += #tAnyParameters.RepetitionFactor;
       #tAnyParameters.RepetitionFactor := 1;
       #tAnyParameters.MemoryAreaAddress := 16#8100_0000 OR (SHL(IN := INT_TO_DWORD(#tOffset), N := 3));
       IF BLKMOV(SRCBLK := #tAny, DSTBLK => #sInData.CompletionStatus) <> 0 THEN
           #sHMI.Status.Error := 1;
           #sHMI.Status.ErrorCode := 1205;
           GOTO Error;
       END_IF;
       #tOffset += #tAnyParameters.RepetitionFactor;
       #tAnyParameters.RepetitionFactor := 1;
       #tAnyParameters.MemoryAreaAddress := 16#8100_0000 OR (SHL(IN := INT_TO_DWORD(#tOffset), N := 3));
       IF BLKMOV(SRCBLK := #tAny, DSTBLK => #sInData.ErrorStatus) <> 0 THEN
           #sHMI.Status.Error := 1;
           #sHMI.Status.ErrorCode := 1205;
           GOTO Error;
       END_IF;
       #tOffset += #tAnyParameters.RepetitionFactor;
       #tAnyParameters.RepetitionFactor := 1;
       #tAnyParameters.MemoryAreaAddress := 16#8100_0000 OR (SHL(IN := INT_TO_DWORD(#tOffset), N := 3));
       IF BLKMOV(SRCBLK := #tAny, DSTBLK => #sInData.TerminalStatus) <> 0 THEN
           #sHMI.Status.Error := 1;
           #sHMI.Status.ErrorCode := 1205;
           GOTO Error;
       END_IF;
       #tOffset += #tAnyParameters.RepetitionFactor;
       #tAnyParameters.RepetitionFactor := 1;
       #tAnyParameters.MemoryAreaAddress := 16#8100_0000 OR (SHL(IN := INT_TO_DWORD(#tOffset), N := 3));
       IF BLKMOV(SRCBLK := #tAny, DSTBLK => #sInData.UnstableReadStatus) <> 0 THEN
           #sHMI.Status.Error := 1;
           #sHMI.Status.ErrorCode := 1205;
           GOTO Error;
       END_IF;
       #tOffset += #tAnyParameters.RepetitionFactor;
       #tAnyParameters.RepetitionFactor := 8;
       #tAnyParameters.MemoryAreaAddress := 16#8100_0000 OR (SHL(IN := INT_TO_DWORD(#tOffset), N := 3));
       IF BLKMOV(SRCBLK := #tAny, DSTBLK => #sInData.MatchingLevelAndTotalEvaluationGradeStatus) <> 0 THEN
           #sHMI.Status.Error := 1;
           #sHMI.Status.ErrorCode := 1205;
           GOTO Error;
       END_IF;
       #tOffset += #tAnyParameters.RepetitionFactor;
       #tAnyParameters.RepetitionFactor := 20;
       #tAnyParameters.MemoryAreaAddress := 16#8100_0000 OR (SHL(IN := INT_TO_DWORD(#tOffset), N := 3));
       IF BLKMOV(SRCBLK := #tAny, DSTBLK => #sInData.OperationResultStatus) <> 0 THEN
           #sHMI.Status.Error := 1;
           #sHMI.Status.ErrorCode := 1205;
           GOTO Error;
       END_IF;
       #tOffset += #tAnyParameters.RepetitionFactor;
       #tAnyParameters.RepetitionFactor := 136;
       #tAnyParameters.MemoryAreaAddress := 16#8100_0000 OR (SHL(IN := INT_TO_DWORD(#tOffset), N := 3));
       IF BLKMOV(SRCBLK := #tAny, DSTBLK => #sInData.ReadData) <> 0 THEN
           #sHMI.Status.Error := 1;
           #sHMI.Status.ErrorCode := 1205;
           GOTO Error;
       END_IF;
   END_REGION ;

   (*Status*)
   REGION Status
       (*Set String length*)
       #sAtCurrentCode[-1] := 128;

       (*Ready*)
       #sHMI.Status.Ready := #iSysRun AND #sCtrl.Sequence = 0
       AND NOT #sInData.BusyStatus.TrggerBusy
       AND NOT #sInData.HandshakeAndGeneralErrorStatus.Error
       AND NOT #sInData.CompletionStatus.ReadComplete
       AND NOT #sInData.ErrorStatus.ReadFailure
       AND NOT #sHMI.Status.Error;//20210605

       (*Busy*)
       #sHMI.Status.Busy := #sInData.BusyStatus.TrggerBusy;

       (*Failure*)
       #sHMI.Status.Failure := #sInData.ErrorStatus.ReadFailure;

       (*Timeout*)
       #sRunTimer(IN := #sCtrl.Sequence <> 0 OR NOT #sHMI.Status.Ready,
                  PT := T#3000MS,
                  Q => #sHMI.Status.TimeOut);
       #sBusyTimer(IN := #sInData.BusyStatus.TrggerBusy,
               PT := T#1000MS,
               Q => #sBusyTimeOut); //20210605

       (*SR1000 Error and Error Code*)    
       IF #sInData.HandshakeAndGeneralErrorStatus.Error THEN
           #sHMI.Status.Error := 1;
           #sHMI.Status.ErrorCode := #sInData.OperationResultStatus.ReadResultCode;
       ELSIF #sHMI.Status.TimeOut THEN
           #sHMI.Status.Error := 1;
           #sHMI.Status.ErrorCode := 1303;
           #sOutData.OperationInstructionControl.ReadRequest := 0; //20210605
       END_IF;



       (*HMI Display*)
       #sHMI.Status.Sequence := #sCtrl.Sequence;

       #sHMI.Indata.ReadComplete := #sInData.CompletionStatus.ReadComplete;
       #sHMI.Indata.ReadFailure := #sInData.ErrorStatus.ReadFailure;
       #sHMI.Indata.GeneralErrorCode := #sInData.OperationResultStatus.GeneralErrorCode;
       #sHMI.Indata.ReadResultCode := #sInData.OperationResultStatus.ReadResultCode;
       #sHMI.Indata.ResultDataSize := #sInData.ReadData.ResultDataSize;

       #sHMI.Outdata.ReadCompleteClear := #sOutData.CompletionClearControl.ReadCompleteClear;
       #sHMI.Outdata.ErrorClear := #sOutData.LatchAndErrorClearControl.ErrorClear;
       #sHMI.Outdata.ReadRequest := #sOutData.OperationInstructionControl.ReadRequest;

   END_REGION ;
   (*Control*)
   REGION Control
       (*Reset command*)
       IF NOT #iSysRun OR (#iManual XOR #sManualOld) OR (#iAuto XOR #sAutoOld) THEN
           #sHMI.Manual.Trigger := 0;
           #ioAutoTrigger := 0;
           #sHMI.Status.iReTriggerTimes := 0;
           #sOutData.OperationInstructionControl.ReadRequest := 0; //20210605
       END_IF;
       #sManualOld := #iManual;
       #sAutoOld := #iAuto;


       //Control Sequece************************************************************************)
       CASE #sCtrl.Sequence OF
           0:(*Trigger*)
               #sOutData.CompletionClearControl.ReadCompleteClear := #sInData.CompletionStatus.ReadComplete;
               IF #sHMI.Status.Ready AND ((#iAuto AND #ioAutoTrigger) XOR (#iManual AND #sHMI.Manual.Trigger)) THEN
                   #sHMI.Status.LastCode := #sHMI.Status.CurrentCode;
                   #sHMI.Status.CurrentCode := '';
                   #sHMI.Status.CurrentLength := 0;
                   #sHMI.Status.ReadOk := 0;
                   #sHMI.Status.ReadNok := 0;
                   #sHMI.Status.Complete := 0;
                   #sOutData.OperationInstructionControl.ReadRequest := 1; //Trigger
                   #sOutData.CompletionClearControl.ReadCompleteClear := 0;
                   #sCtrl.Sequence := 1;
               ELSE
                   #sOutData.OperationInstructionControl.ReadRequest := 0;
               END_IF;
           1:(*Reading*)
               IF NOT #sInData.HandshakeAndGeneralErrorStatus.Error
                   AND #sOutData.OperationInstructionControl.ReadRequest
                   AND #sInData.BusyStatus.TrggerBusy THEN
                   #sHMI.Status.iReTriggerTimes := #sHMI.Status.iReTriggerTimes + 1;
                   //#sHMI.Manual.Trigger := 0;
                   #sCtrl.Sequence := 2;
               END_IF;
           2:(*Complete*)
               IF (NOT #sInData.HandshakeAndGeneralErrorStatus.Error AND NOT #sInData.BusyStatus.TrggerBusy AND #sInData.CompletionStatus.ReadComplete)
                   OR #sBusyTimeOut THEN
                   #sOutData.OperationInstructionControl.ReadRequest := 0;
                   #sCtrl.Sequence := 3;
               END_IF;
           3:(*Result*)
               IF NOT #sInData.HandshakeAndGeneralErrorStatus.Error
                   AND NOT #sOutData.OperationInstructionControl.ReadRequest
                   AND #sInData.CompletionStatus.ReadComplete
                   AND #sInData.ReadData.ResultDataSize <= 128
                   AND #sInData.ReadData.ResultDataSize > 0 THEN
                   Chars_TO_Strg(Chars := #sInData.ReadData.ResultData,
                                 pChars := 0, //20210605
                                 Cnt := #sInData.ReadData.ResultDataSize,
                                 Strg => #sCurrentCode);

                   #sFindCurrentPos  :=  FIND(IN1 := #sCurrentCode, IN2 := '$R');

                   #sCurrentCode := DELETE(IN := #sCurrentCode, L := 2, P := #sFindCurrentPos);

                   #sHMI.Status.CurrentCode := #sCurrentCode;
                   IF #sHMI.Status.CurrentCode = 'ERROR' OR #sInData.ErrorStatus.ReadFailure THEN
                       #sCtrl.Sequence := 4;
                   ELSE
                       #sHMI.Status.ReadOk := 1;
                       #sHMI.Status.ReadNok := 0;
                       #sCtrl.Sequence := 5;
                   END_IF;
               END_IF;

           4: (*ReTrigger*)
               IF #sHMI.Status.iReTriggerTimes < #iReTriggerLimitTimes THEN
                   #sOutData.CompletionClearControl.ReadCompleteClear := 1;
                   IF NOT #sInData.CompletionStatus.ReadComplete AND NOT #sInData.ErrorStatus.ReadFailure THEN
                       #sCtrl.Sequence := 0;
                   END_IF;
               ELSE
                   #sHMI.Status.ReadOk := 0;
                   #sHMI.Status.ReadNok := 1;
                   #sCtrl.Sequence := 5;
               END_IF;

           5:(*Clear*)
               IF NOT #sOutData.OperationInstructionControl.ReadRequest
                   AND #sInData.CompletionStatus.ReadComplete THEN
                   #sOutData.CompletionClearControl.ReadCompleteClear := 1;
               ELSE
                   #sOutData.CompletionClearControl.ReadCompleteClear := 0;
                   #ioAutoTrigger := 0;
                   #sHMI.Manual.Trigger := 0;
                   #sHMI.Status.iReTriggerTimes := 0;
                   #sHMI.Status.Complete := 1;
                   #sCtrl.Sequence := 0;
               END_IF;
           ELSE(*Limit*)
               #sCtrl.Sequence := 0;
       END_CASE;
   END_REGION ;

   REGION Reset
   IF (#sHMI.Status.Error OR #sHMI.Status.Failure OR #sHMI.Status.TimeOut) THEN
       IF #iReset THEN
           #sOutData.LatchAndErrorClearControl.ErrorClear := 1;
           #sOutData.OperationInstructionControl.ReadRequest := 0;
           #ioAutoTrigger := 0;
           #sHMI.Manual.Trigger := 0;
           #sCtrl.Sequence := 0;
           #sHMI.Status.Error := 0;
           #sHMI.Status.ErrorCode := 0;
       END_IF;
   ELSE
       #sOutData.LatchAndErrorClearControl.ErrorClear := 0;
   END_IF;
   END_REGION ;


   (*Write Data from PLC memory to KEYENCE SR-1000*)
   REGION Write outputs
       #tAnyParameters.SyntaxID := 16#10;
       #tAnyParameters.DataType := 16#02;
       #tOffset := #iO_Address;
       #tAnyParameters.RepetitionFactor := 1;
       #tAnyParameters.DB_Number := 16#0;
       #tAnyParameters.MemoryAreaAddress := 16#8200_0000 OR (SHL(IN := INT_TO_DWORD(#tOffset), N := 3)); //B#16#82 Output Area
       IF BLKMOV(SRCBLK := #sOutData.LatchAndErrorClearControl, DSTBLK => #tAny) <> 0 THEN
           #sHMI.Status.Error := 1;
           #sHMI.Status.ErrorCode := 1206;
           GOTO Error;
       END_IF;
       #tOffset += #tAnyParameters.RepetitionFactor;
       #tAnyParameters.RepetitionFactor := 1;
       #tAnyParameters.MemoryAreaAddress := 16#8200_0000 OR (SHL(IN := INT_TO_DWORD(#tOffset), N := 3));
       IF BLKMOV(SRCBLK := #sOutData.OperationInstructionControl, DSTBLK => #tAny) <> 0 THEN
           #sHMI.Status.Error := 1;
           #sHMI.Status.ErrorCode := 1206;
           GOTO Error;
       END_IF;
       #tOffset += #tAnyParameters.RepetitionFactor;
       #tAnyParameters.RepetitionFactor := 1;
       #tAnyParameters.MemoryAreaAddress := 16#8200_0000 OR (SHL(IN := INT_TO_DWORD(#tOffset), N := 3));
       IF BLKMOV(SRCBLK := #sOutData.CompletionClearControl, DSTBLK => #tAny) <> 0 THEN
           #sHMI.Status.Error := 1;
           #sHMI.Status.ErrorCode := 1206;
           GOTO Error;
       END_IF;
       #tOffset += #tAnyParameters.RepetitionFactor;
       #tAnyParameters.RepetitionFactor := 2;
       #tAnyParameters.MemoryAreaAddress := 16#8200_0000 OR (SHL(IN := INT_TO_DWORD(#tOffset), N := 3));
       IF BLKMOV(SRCBLK := #sOutData.ParameterBankNumber, DSTBLK => #tAny) <> 0 THEN
           #sHMI.Status.Error := 1;
           #sHMI.Status.ErrorCode := 1206;
           GOTO Error;
       END_IF;
       #tOffset += #tAnyParameters.RepetitionFactor;
       #tAnyParameters.RepetitionFactor := 130;
       #tAnyParameters.MemoryAreaAddress := 16#8200_0000 OR (SHL(IN := INT_TO_DWORD(#tOffset), N := 3));
       IF BLKMOV(SRCBLK := #sOutData.UserData, DSTBLK => #tAny) <> 0 THEN
           #sHMI.Status.Error := 1;
           #sHMI.Status.ErrorCode := 1206;
           GOTO Error;
       END_IF;

   //FB OUTPUT    
       #oReady := #sHMI.Status.Ready;
       #oComplete := #sHMI.Status.Complete;
       #oError := #sHMI.Status.Error;
       #oErrorCode := #sHMI.Status.ErrorCode;

   END_REGION ;
   (*The end of the function block*)
   REGION End function
       ENO := 1;
       RETURN;
   Error:
       #sHMI.Status.Ready := 0;
       #tEmpty := 16#0000_0000;
       #tRetVal := FILL(BVAL := #tEmpty, BLK => #sOutData.LatchAndErrorClearControl);
       #tRetVal := FILL(BVAL := #tEmpty, BLK => #sOutData.OperationInstructionControl);
       #tRetVal := FILL(BVAL := #tEmpty, BLK => #sOutData.CompletionClearControl);
       #tRetVal := FILL(BVAL := #tEmpty, BLK => #sOutData.ParameterBankNumber);
       #tRetVal := FILL(BVAL := #tEmpty, BLK => #sOutData.UserData);
       ENO := 0;
       RETURN;
   END_REGION ;
END_FUNCTION_BLOCK

FUNCTION "Servo" : Void   // FC2500, LAD
{ S7_Optimized_Access := 'TRUE' }
// stored: AutoNumber false, SetENOAutomatically false
BEGIN

REGION Network 1
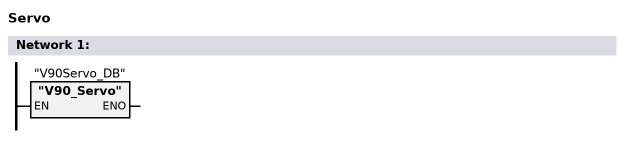
   RUNG wire#powerrail
      "V90Servo_DB"()
   END_RUNG
   // the same network as SCL:
   "V90Servo_DB"();   // "V90_Servo"
END_REGION
END_FUNCTION

FUNCTION_BLOCK "V90_Servo"   // FB2500, LAD
{ S7_Optimized_Access := 'TRUE' }
// stored: AutoNumber false, MemoryReserve 100, SetENOAutomatically false
   VAR
      Servo_380A1 { S7_SetPoint := 'True'} : "fbV90Ctrl";   // *
      Servo_381A1 { S7_SetPoint := 'True'} : "fbV90Ctrl";   // *
      Servo_382A1 { S7_SetPoint := 'True'} : "fbV90Ctrl";   // *
      Servo_383A1 { S7_SetPoint := 'True'} : "fbV90Ctrl";   // *
      Servo1 { S7_SetPoint := 'True'} : "SevroStart&PosCheck";
      Servo2 { S7_SetPoint := 'True'} : "SevroStart&PosCheck";
      Servo3 { S7_SetPoint := 'True'} : "SevroStart&PosCheck";
      Servo4 { S7_SetPoint := 'True'} : "SevroStart&PosCheck";
      Servo2SafetyPos { S7_SetPoint := 'True'} : DInt;
      Servo4SafetyPos { S7_SetPoint := 'True'} : DInt;
      IEC_Timer_0_Instance { S7_SetPoint := 'True'} : TON_TIME;
      P { S7_SetPoint := 'True'} : Array[0..10] of Bool;
   END_VAR
   VAR_TEMP
      Sevro1ActPos : Real;
      Sevro1StartList : Bool;
      Sevro2ActPos : Real;
      Sevro2StartList : Bool;
      Sevro3ActPos : Real;
      Sevro3StartList : Bool;
      Sevro4ActPos : Real;
      Sevro4StartList : Bool;
   END_VAR
   VAR_TEMP   // added for the SCL form of the ladder/FBD networks
      _w1 : Bool;
      _w2 : Bool;
   END_VAR
BEGIN

REGION Network 1: <<<<<<<<<<<<<<<<<<<<<380A1 Servo>>>>>>>>>>>>>>>>>>>>>>>>>
END_REGION

REGION Network 2: negtive motion/action/...automaticly
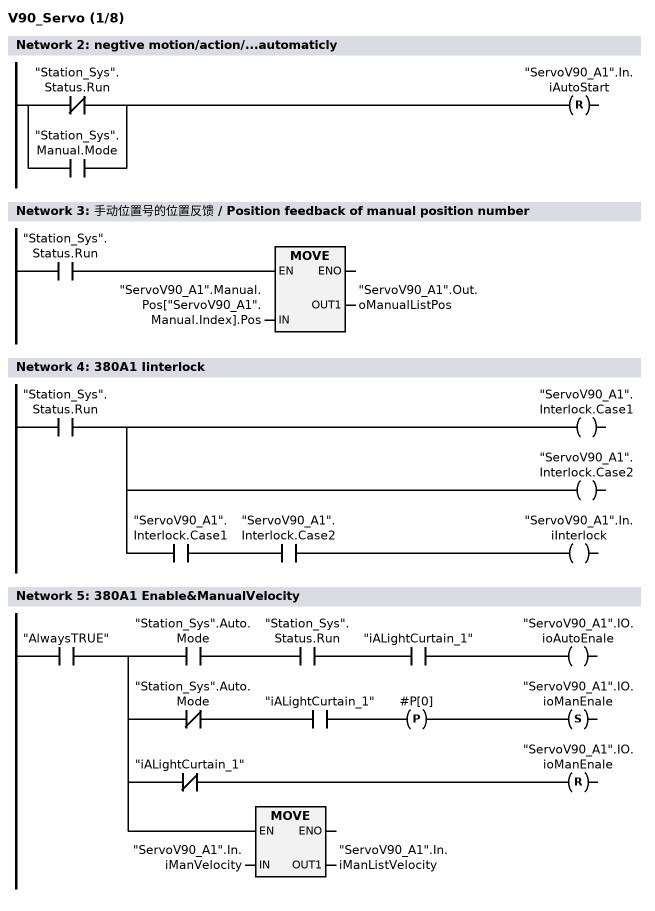
   RUNG wire#powerrail
      I_Contact( "Station_Sys".Status.Run )
      wire#w1
      R_Coil( "ServoV90_A1".In.iAutoStart )
   END_RUNG
   RUNG wire#powerrail
      Contact( "Station_Sys".Manual.Mode )
   END_RUNG wire#w1
   // the same network as SCL:
   IF NOT "Station_Sys".Status.Run OR "Station_Sys".Manual.Mode THEN
       "ServoV90_A1".In.iAutoStart := FALSE;
   END_IF;
END_REGION

REGION Network 3: 手动位置号的位置反馈 / Position feedback of manual position number
   RUNG wire#powerrail
      Contact( "Station_Sys".Status.Run )
      Move(in := "ServoV90_A1".Manual.Pos["ServoV90_A1".Manual.Index].Pos, out1 => "ServoV90_A1".Out.oManualListPos)
   END_RUNG
   // the same network as SCL:
   IF "Station_Sys".Status.Run THEN
       "ServoV90_A1".Out.oManualListPos := "ServoV90_A1".Manual.Pos["ServoV90_A1".Manual.Index].Pos;
   END_IF;
END_REGION

REGION Network 4: 380A1 Iinterlock
   RUNG wire#powerrail
      Contact( "Station_Sys".Status.Run )
      wire#w1
      Coil( "ServoV90_A1".Interlock.Case1 )
   END_RUNG
   RUNG wire#w1
      Coil( "ServoV90_A1".Interlock.Case2 )
   END_RUNG
   RUNG wire#w1
      Contact( "ServoV90_A1".Interlock.Case1 )
      Contact( "ServoV90_A1".Interlock.Case2 )
      Coil( "ServoV90_A1".In.iInterlock )
   END_RUNG
   // the same network as SCL:
   "ServoV90_A1".Interlock.Case1 := "Station_Sys".Status.Run;
   "ServoV90_A1".Interlock.Case2 := "Station_Sys".Status.Run;
   "ServoV90_A1".In.iInterlock := "Station_Sys".Status.Run AND "ServoV90_A1".Interlock.Case1 AND "ServoV90_A1".Interlock.Case2;
END_REGION

REGION Network 5: 380A1 Enable&ManualVelocity
   RUNG wire#powerrail
      Contact( "AlwaysTRUE" )
      wire#w1
      Contact( "Station_Sys".Auto.Mode )
      Contact( "Station_Sys".Status.Run )
      Contact( "iALightCurtain_1" )
      Coil( "ServoV90_A1".IO.ioAutoEnale )
   END_RUNG
   RUNG wire#w1
      I_Contact( "Station_Sys".Auto.Mode )
      Contact( "iALightCurtain_1" )
      P_Trig( #P[0] )
      S_Coil( "ServoV90_A1".IO.ioManEnale )
   END_RUNG
   RUNG wire#w1
      I_Contact( "iALightCurtain_1" )
      R_Coil( "ServoV90_A1".IO.ioManEnale )
   END_RUNG
   RUNG wire#w1
      Move(in := "ServoV90_A1".In.iManVelocity, out1 => "ServoV90_A1".In.iManListVelocity)
   END_RUNG
   // the same network as SCL:
   "ServoV90_A1".IO.ioAutoEnale := "AlwaysTRUE" AND "Station_Sys".Auto.Mode AND "Station_Sys".Status.Run AND "iALightCurtain_1";
   #_w1 := "AlwaysTRUE" AND NOT "Station_Sys".Auto.Mode AND "iALightCurtain_1";
   #_w2 := #_w1 AND NOT #P[0];   // rising edge
   #P[0] := #_w1;
   IF #_w2 THEN "ServoV90_A1".IO.ioManEnale := TRUE; END_IF;
   IF "AlwaysTRUE" AND NOT "iALightCurtain_1" THEN "ServoV90_A1".IO.ioManEnale := FALSE; END_IF;
   IF "AlwaysTRUE" THEN "ServoV90_A1".In.iManListVelocity := "ServoV90_A1".In.iManVelocity; END_IF;
END_REGION

REGION Network 6 (SCL): 380A1 RecipePosition
    IF "Station_Sys".Status.Run THEN
        "ServoV90_A1".Manual.Pos[1].Pos := "ServoV90_A1".Auto.Pos[1].Pos :=REAL_TO_DINT("Parameter".AxisRun.Axis[1].Pos1.Position*1000);
        "ServoV90_A1".Manual.Pos[1].Vel := "ServoV90_A1".Auto.Pos[1].Vel := "Parameter".AxisRun.Axis[1].Pos1.Speed;

        "ServoV90_A1".Manual.Pos[2].Pos := "ServoV90_A1".Auto.Pos[2].Pos := REAL_TO_DINT("Parameter".AxisRun.Axis[1].Pos2.Position*1000);
       "ServoV90_A1".Manual.Pos[2].Vel := "ServoV90_A1".Auto.Pos[2].Vel := "Parameter".AxisRun.Axis[1].Pos2.Speed;

       "ServoV90_A1".Manual.Pos[3].Pos := "ServoV90_A1".Auto.Pos[3].Pos := REAL_TO_DINT("Parameter".AxisRun.Axis[1].Pos3.Position*1000);
       "ServoV90_A1".Manual.Pos[3].Vel := "ServoV90_A1".Auto.Pos[3].Vel := "Parameter".AxisRun.Axis[1].Pos3.Speed;

       "ServoV90_A1".Manual.Pos[4].Pos := "ServoV90_A1".Auto.Pos[4].Pos := REAL_TO_DINT("Parameter".AxisRun.Axis[1].Pos4.Position*1000);
       "ServoV90_A1".Manual.Pos[4].Vel := "ServoV90_A1".Auto.Pos[4].Vel := "Parameter".AxisRun.Axis[1].Pos4.Speed;

       "ServoV90_A1".Manual.Pos[5].Pos := "ServoV90_A1".Auto.Pos[5].Pos := REAL_TO_DINT("Parameter".AxisRun.Axis[1].Pos5.Position*1000);
       "ServoV90_A1".Manual.Pos[5].Vel := "ServoV90_A1".Auto.Pos[5].Vel := "Parameter".AxisRun.Axis[1].Pos5.Speed;

       "ServoV90_A1".Manual.Pos[6].Pos := "ServoV90_A1".Auto.Pos[6].Pos := REAL_TO_DINT("Parameter".AxisRun.Axis[1].Pos6.Position*1000);
       "ServoV90_A1".Manual.Pos[6].Vel := "ServoV90_A1".Auto.Pos[6].Vel := "Parameter".AxisRun.Axis[1].Pos6.Speed;

       "ServoV90_A1".Manual.Pos[7].Pos := "ServoV90_A1".Auto.Pos[7].Pos := REAL_TO_DINT("Parameter".AxisRun.Axis[1].Pos7.Position*1000);
       "ServoV90_A1".Manual.Pos[7].Vel := "ServoV90_A1".Auto.Pos[7].Vel := "Parameter".AxisRun.Axis[1].Pos7.Speed;

       "ServoV90_A1".Manual.Pos[8].Pos := "ServoV90_A1".Auto.Pos[8].Pos := REAL_TO_DINT("Parameter".AxisRun.Axis[1].Pos8.Position*1000);
       "ServoV90_A1".Manual.Pos[8].Vel := "ServoV90_A1".Auto.Pos[8].Vel := "Parameter".AxisRun.Axis[1].Pos8.Speed;

       "ServoV90_A1".Manual.Pos[9].Pos := "ServoV90_A1".Auto.Pos[9].Pos := REAL_TO_DINT("Parameter".AxisRun.Axis[1].Pos9.Position*1000);
       "ServoV90_A1".Manual.Pos[9].Vel := "ServoV90_A1".Auto.Pos[9].Vel := "Parameter".AxisRun.Axis[1].Pos9.Speed;

   END_IF;
END_REGION

